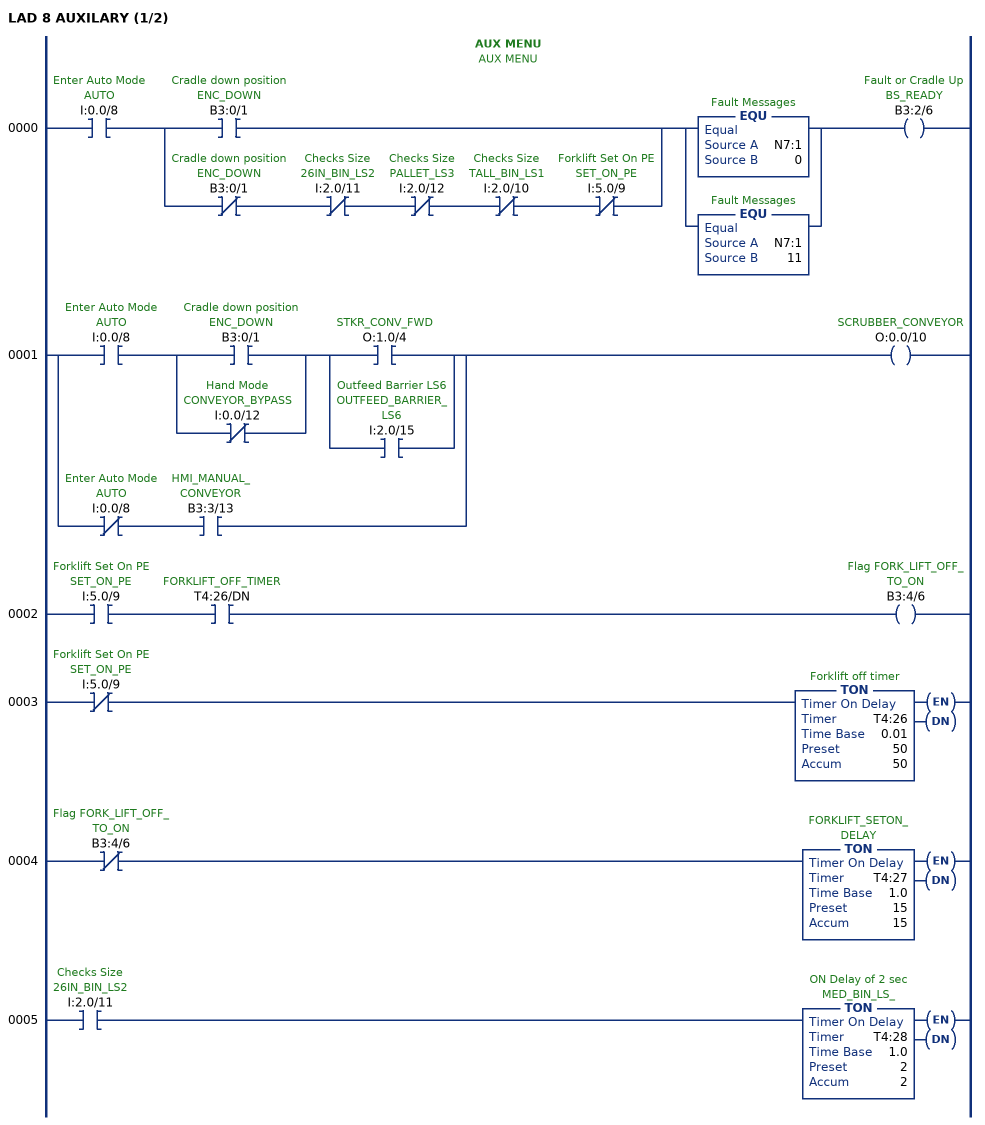
% Rung: 0 %
% TITLE: AUX MENU %
% AUX MENU %
SOR XIC I:0.0/8 BST XIC B3:0/1 NXB XIO B3:0/1 XIO I:2.0/11 XIO I:2.0/12 XIO I:2.0/10 XIO I:5.0/9 BND BST EQU N7:1 0 NXB EQU N7:1 11 BND OTE B3:2/6 EOR
%   I:0.0/8  AUTO  "Enter Auto Mode" %
%   B3:0/1  ENC_DOWN  "Cradle down position" %
%   I:2.0/11  26IN_BIN_LS2  "Checks Size" %
%   I:2.0/12  PALLET_LS3  "Checks Size" %
%   I:2.0/10  TALL_BIN_LS1  "Checks Size" %
%   I:5.0/9  SET_ON_PE  "Forklift Set On PE" %
%   N7:1  "Fault Messages" %
%   B3:2/6  BS_READY  "Fault or Cradle Up" %
% Rung: 1 %
SOR BST XIC I:0.0/8 BST XIC B3:0/1 NXB XIO I:0.0/12 BND BST XIC O:1.0/4 NXB XIC I:2.0/15 BND NXB XIO I:0.0/8 XIC B3:3/13 BND OTE O:0.0/10 EOR
%   I:0.0/8  AUTO  "Enter Auto Mode" %
%   B3:0/1  ENC_DOWN  "Cradle down position" %
%   I:0.0/12  CONVEYOR_BYPASS  "Hand Mode" %
%   O:1.0/4  STKR_CONV_FWD %
%   I:2.0/15  OUTFEED_BARRIER_LS6  "Outfeed Barrier LS6" %
%   B3:3/13  HMI_MANUAL_CONVEYOR %
%   O:0.0/10  SCRUBBER_CONVEYOR %
% Rung: 2 %
SOR XIC I:5.0/9 XIC T4:26/DN OTE B3:4/6 EOR
%   I:5.0/9  SET_ON_PE  "Forklift Set On PE" %
%   T4:26/DN  FORKLIFT_OFF_TIMER %
%   B3:4/6  FORK_LIFT_OFF_TO_ON  "Flag" %
% Rung: 3 %
SOR XIO I:5.0/9 TON T4:26 0.01 50 50 EOR
%   I:5.0/9  SET_ON_PE  "Forklift Set On PE" %
%   T4:26  "Forklift off timer" %
% Rung: 4 %
SOR XIO B3:4/6 TON T4:27 1.0 15 15 EOR
%   B3:4/6  FORK_LIFT_OFF_TO_ON  "Flag" %
%   T4:27  FORKLIFT_SETON_DELAY %
% Rung: 5 %
SOR XIC I:2.0/11 TON T4:28 1.0 2 2 EOR
%   I:2.0/11  26IN_BIN_LS2  "Checks Size" %
%   T4:28  MED_BIN_LS_  "ON Delay of 2 sec" %

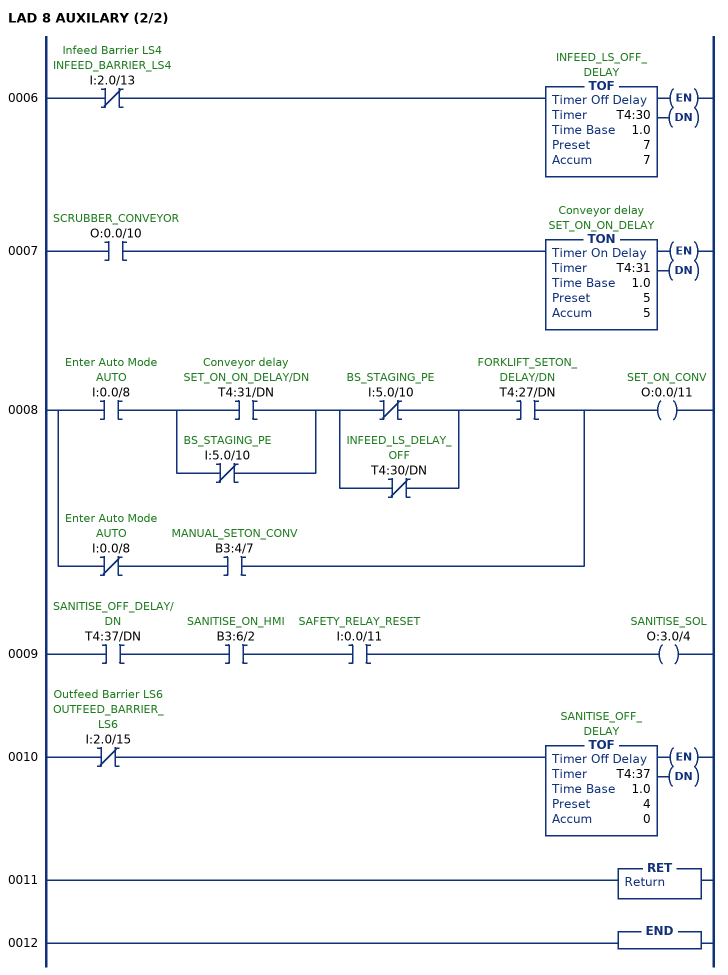
% Rung: 6 %
SOR XIO I:2.0/13 TOF T4:30 1.0 7 7 EOR
%   I:2.0/13  INFEED_BARRIER_LS4  "Infeed Barrier LS4" %
%   T4:30  INFEED_LS_OFF_DELAY %
% Rung: 7 %
SOR XIC O:0.0/10 TON T4:31 1.0 5 5 EOR
%   O:0.0/10  SCRUBBER_CONVEYOR %
%   T4:31  SET_ON_ON_DELAY  "Conveyor delay" %
% Rung: 8 %
SOR BST XIC I:0.0/8 BST XIC T4:31/DN NXB XIO I:5.0/10 BND BST XIO I:5.0/10 NXB XIO T4:30/DN BND XIC T4:27/DN NXB XIO I:0.0/8 XIC B3:4/7 BND OTE O:0.0/11 EOR
%   I:0.0/8  AUTO  "Enter Auto Mode" %
%   T4:31  SET_ON_ON_DELAY  "Conveyor delay" %
%   I:5.0/10  BS_STAGING_PE %
%   T4:30/DN  INFEED_LS_DELAY_OFF %
%   T4:27  FORKLIFT_SETON_DELAY %
%   B3:4/7  MANUAL_SETON_CONV %
%   O:0.0/11  SET_ON_CONV %
% Rung: 9 %
SOR XIC T4:37/DN XIC B3:6/2 XIC I:0.0/11 OTE O:3.0/4 EOR
%   T4:37  SANITISE_OFF_DELAY %
%   B3:6/2  SANITISE_ON_HMI %
%   I:0.0/11  SAFETY_RELAY_RESET %
%   O:3.0/4  SANITISE_SOL %
% Rung: 10 %
SOR XIO I:2.0/15 TOF T4:37 1.0 4 0 EOR
%   I:2.0/15  OUTFEED_BARRIER_LS6  "Outfeed Barrier LS6" %
%   T4:37  SANITISE_OFF_DELAY %
% Rung: 11 %
SOR RET EOR
% Rung: 12 %
SOR END EOR

LADDER 9 "FAULTS"
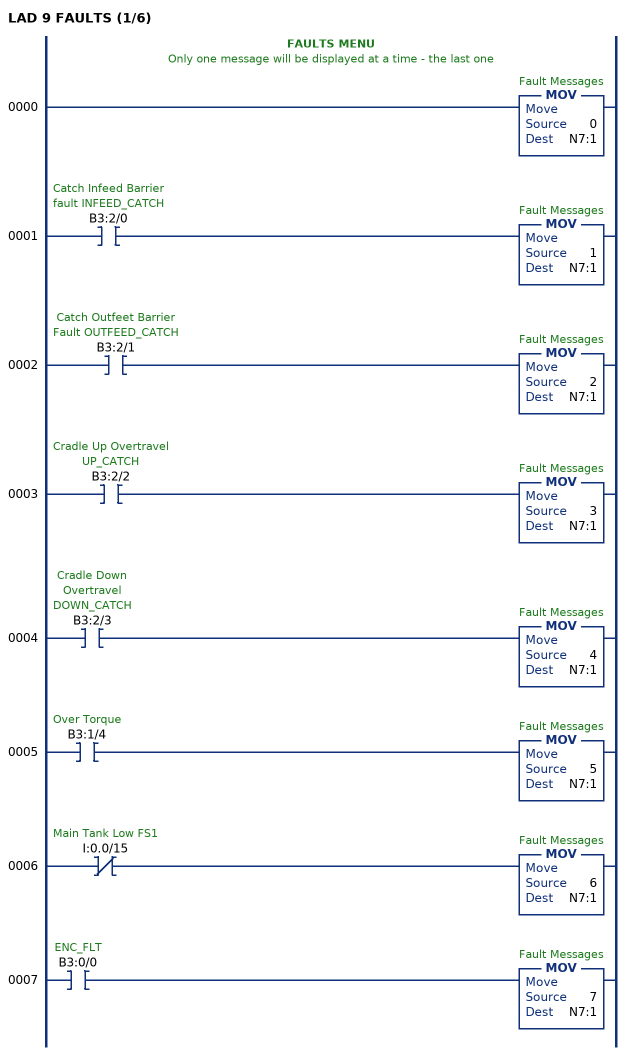
% Rung: 0 %
% TITLE: FAULTS MENU %
% Only one message will be displayed at a time - the last one %
SOR MOV 0 N7:1 EOR
%   N7:1  "Fault Messages" %
% Rung: 1 %
SOR XIC B3:2/0 MOV 1 N7:1 EOR
%   B3:2/0  INFEED_CATCH  "Catch Infeed Barrier fault" %
%   N7:1  "Fault Messages" %
% Rung: 2 %
SOR XIC B3:2/1 MOV 2 N7:1 EOR
%   B3:2/1  OUTFEED_CATCH  "Catch Outfeet Barrier Fault" %
%   N7:1  "Fault Messages" %
% Rung: 3 %
SOR XIC B3:2/2 MOV 3 N7:1 EOR
%   B3:2/2  UP_CATCH  "Cradle Up Overtravel" %
%   N7:1  "Fault Messages" %
% Rung: 4 %
SOR XIC B3:2/3 MOV 4 N7:1 EOR
%   B3:2/3  DOWN_CATCH  "Cradle Down Overtravel" %
%   N7:1  "Fault Messages" %
% Rung: 5 %
SOR XIC B3:1/4 MOV 5 N7:1 EOR
%   B3:1/4  "Over Torque" %
%   N7:1  "Fault Messages" %
% Rung: 6 %
SOR XIO I:0.0/15 MOV 6 N7:1 EOR
%   I:0.0/15  FS1  "Main Tank Low" %
%   N7:1  "Fault Messages" %
% Rung: 7 %
SOR XIC B3:0/0 MOV 7 N7:1 EOR
%   B3:0/0  ENC_FLT %
%   N7:1  "Fault Messages" %

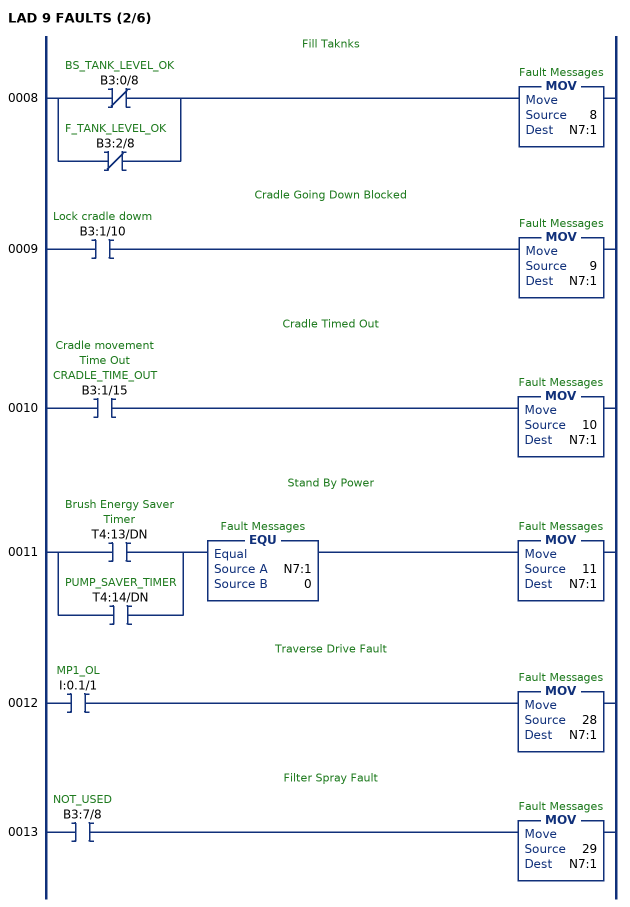
% Rung: 8 %
% Fill Taknks %
SOR BST XIO B3:0/8 NXB XIO B3:2/8 BND MOV 8 N7:1 EOR
%   B3:0/8  BS_TANK_LEVEL_OK %
%   B3:2/8  F_TANK_LEVEL_OK %
%   N7:1  "Fault Messages" %
% Rung: 9 %
% Cradle Going Down Blocked %
SOR XIC B3:1/10 MOV 9 N7:1 EOR
%   B3:1/10  "Lock cradle dowm" %
%   N7:1  "Fault Messages" %
% Rung: 10 %
% Cradle Timed Out %
SOR XIC B3:1/15 MOV 10 N7:1 EOR
%   B3:1/15  CRADLE_TIME_OUT  "Cradle movement Time Out" %
%   N7:1  "Fault Messages" %
% Rung: 11 %
% Stand By Power %
SOR BST XIC T4:13/DN NXB XIC T4:14/DN BND EQU N7:1 0 MOV 11 N7:1 EOR
%   T4:13  "Brush Energy Saver Timer" %
%   T4:14/DN  PUMP_SAVER_TIMER %
%   N7:1  "Fault Messages" %
% Rung: 12 %
% Traverse Drive Fault %
SOR XIC I:0.1/1 MOV 28 N7:1 EOR
%   I:0.1/1  MP1_OL %
%   N7:1  "Fault Messages" %
% Rung: 13 %
% Filter Spray Fault %
SOR XIC B3:7/8 MOV 29 N7:1 EOR
%   B3:7/8  NOT_USED %
%   N7:1  "Fault Messages" %

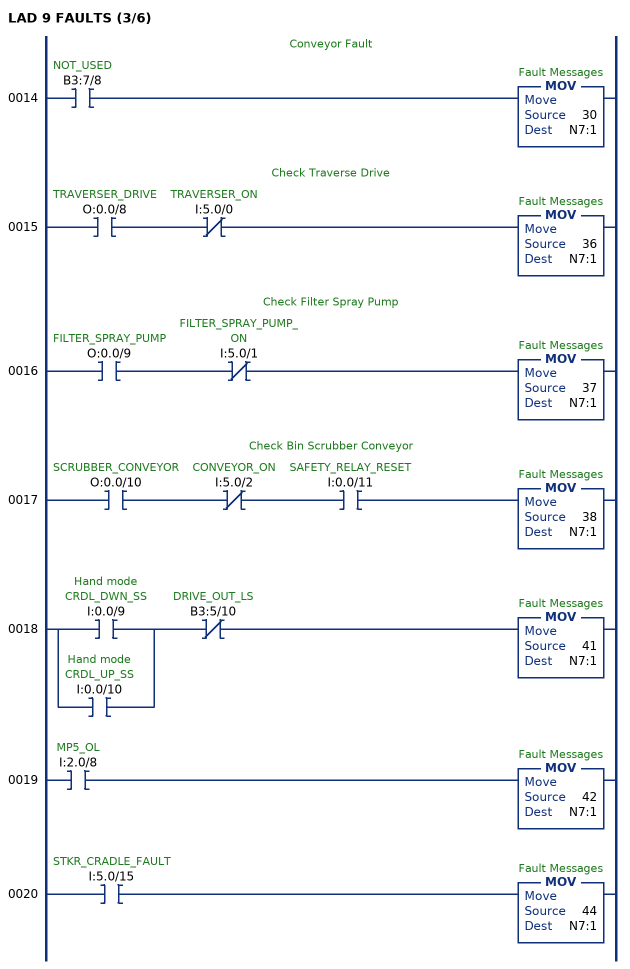
% Rung: 14 %
% Conveyor Fault %
SOR XIC B3:7/8 MOV 30 N7:1 EOR
%   B3:7/8  NOT_USED %
%   N7:1  "Fault Messages" %
% Rung: 15 %
% Check Traverse Drive %
SOR XIC O:0.0/8 XIO I:5.0/0 MOV 36 N7:1 EOR
%   O:0.0/8  TRAVERSER_DRIVE %
%   I:5.0/0  TRAVERSER_ON %
%   N7:1  "Fault Messages" %
% Rung: 16 %
% Check Filter Spray Pump %
SOR XIC O:0.0/9 XIO I:5.0/1 MOV 37 N7:1 EOR
%   O:0.0/9  FILTER_SPRAY_PUMP %
%   I:5.0/1  FILTER_SPRAY_PUMP_ON %
%   N7:1  "Fault Messages" %
% Rung: 17 %
% Check Bin Scrubber Conveyor %
SOR XIC O:0.0/10 XIO I:5.0/2 XIC I:0.0/11 MOV 38 N7:1 EOR
%   O:0.0/10  SCRUBBER_CONVEYOR %
%   I:5.0/2  CONVEYOR_ON %
%   I:0.0/11  SAFETY_RELAY_RESET %
%   N7:1  "Fault Messages" %
% Rung: 18 %
SOR BST XIC I:0.0/9 NXB XIC I:0.0/10 BND XIO B3:5/10 MOV 41 N7:1 EOR
%   I:0.0/9  CRDL_DWN_SS  "Hand mode" %
%   I:0.0/10  CRDL_UP_SS  "Hand mode" %
%   B3:5/10  DRIVE_OUT_LS %
%   N7:1  "Fault Messages" %
% Rung: 19 %
SOR XIC I:2.0/8 MOV 42 N7:1 EOR
%   I:2.0/8  MP5_OL %
%   N7:1  "Fault Messages" %
% Rung: 20 %
SOR XIC I:5.0/15 MOV 44 N7:1 EOR
%   I:5.0/15  STKR_CRADLE_FAULT %
%   N7:1  "Fault Messages" %

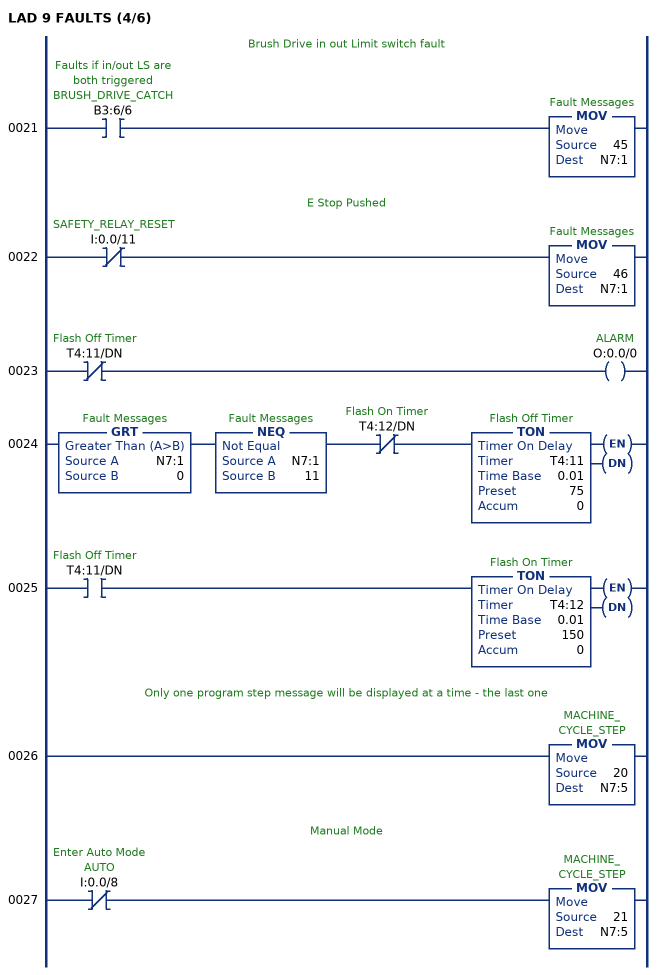
% Rung: 21 %
% Brush Drive in out Limit switch fault %
SOR XIC B3:6/6 MOV 45 N7:1 EOR
%   B3:6/6  BRUSH_DRIVE_CATCH  "Faults if in/out LS are both triggered" %
%   N7:1  "Fault Messages" %
% Rung: 22 %
% E Stop Pushed %
SOR XIO I:0.0/11 MOV 46 N7:1 EOR
%   I:0.0/11  SAFETY_RELAY_RESET %
%   N7:1  "Fault Messages" %
% Rung: 23 %
SOR XIO T4:11/DN OTE O:0.0/0 EOR
%   T4:11  "Flash Off Timer" %
%   O:0.0/0  ALARM %
% Rung: 24 %
SOR GRT N7:1 0 NEQ N7:1 11 XIO T4:12/DN TON T4:11 0.01 75 0 EOR
%   N7:1  "Fault Messages" %
%   T4:12  "Flash On Timer" %
%   T4:11  "Flash Off Timer" %
% Rung: 25 %
SOR XIC T4:11/DN TON T4:12 0.01 150 0 EOR
%   T4:11  "Flash Off Timer" %
%   T4:12  "Flash On Timer" %
% Rung: 26 %
% Only one program step message will be displayed at a time - the last one %
SOR MOV 20 N7:5 EOR
%   N7:5  MACHINE_CYCLE_STEP %
% Rung: 27 %
% Manual Mode %
SOR XIO I:0.0/8 MOV 21 N7:5 EOR
%   I:0.0/8  AUTO  "Enter Auto Mode" %
%   N7:5  MACHINE_CYCLE_STEP %

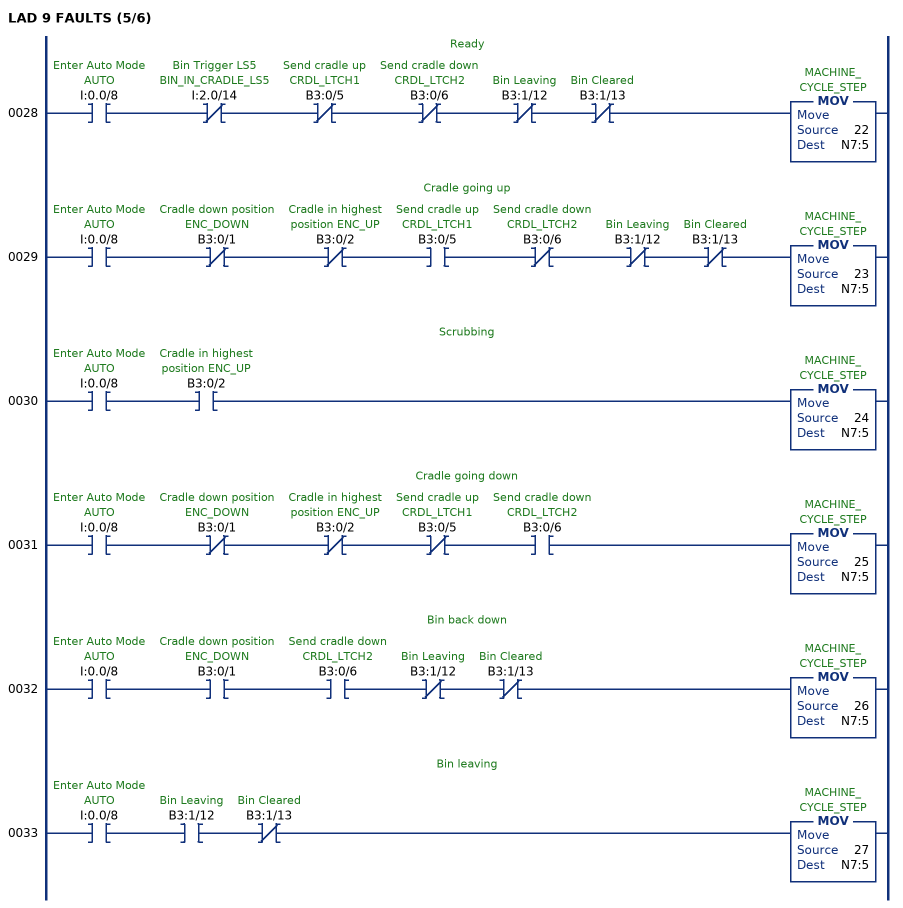
% Rung: 28 %
% Ready %
SOR XIC I:0.0/8 XIO I:2.0/14 XIO B3:0/5 XIO B3:0/6 XIO B3:1/12 XIO B3:1/13 MOV 22 N7:5 EOR
%   I:0.0/8  AUTO  "Enter Auto Mode" %
%   I:2.0/14  BIN_IN_CRADLE_LS5  "Bin Trigger LS5" %
%   B3:0/5  CRDL_LTCH1  "Send cradle up" %
%   B3:0/6  CRDL_LTCH2  "Send cradle down" %
%   B3:1/12  "Bin Leaving" %
%   B3:1/13  "Bin Cleared" %
%   N7:5  MACHINE_CYCLE_STEP %
% Rung: 29 %
% Cradle going up %
SOR XIC I:0.0/8 XIO B3:0/1 XIO B3:0/2 XIC B3:0/5 XIO B3:0/6 XIO B3:1/12 XIO B3:1/13 MOV 23 N7:5 EOR
%   I:0.0/8  AUTO  "Enter Auto Mode" %
%   B3:0/1  ENC_DOWN  "Cradle down position" %
%   B3:0/2  ENC_UP  "Cradle in highest position" %
%   B3:0/5  CRDL_LTCH1  "Send cradle up" %
%   B3:0/6  CRDL_LTCH2  "Send cradle down" %
%   B3:1/12  "Bin Leaving" %
%   B3:1/13  "Bin Cleared" %
%   N7:5  MACHINE_CYCLE_STEP %
% Rung: 30 %
% Scrubbing %
SOR XIC I:0.0/8 XIC B3:0/2 MOV 24 N7:5 EOR
%   I:0.0/8  AUTO  "Enter Auto Mode" %
%   B3:0/2  ENC_UP  "Cradle in highest position" %
%   N7:5  MACHINE_CYCLE_STEP %
% Rung: 31 %
% Cradle going down %
SOR XIC I:0.0/8 XIO B3:0/1 XIO B3:0/2 XIO B3:0/5 XIC B3:0/6 MOV 25 N7:5 EOR
%   I:0.0/8  AUTO  "Enter Auto Mode" %
%   B3:0/1  ENC_DOWN  "Cradle down position" %
%   B3:0/2  ENC_UP  "Cradle in highest position" %
%   B3:0/5  CRDL_LTCH1  "Send cradle up" %
%   B3:0/6  CRDL_LTCH2  "Send cradle down" %
%   N7:5  MACHINE_CYCLE_STEP %
% Rung: 32 %
% Bin back down %
SOR XIC I:0.0/8 XIC B3:0/1 XIC B3:0/6 XIO B3:1/12 XIO B3:1/13 MOV 26 N7:5 EOR
%   I:0.0/8  AUTO  "Enter Auto Mode" %
%   B3:0/1  ENC_DOWN  "Cradle down position" %
%   B3:0/6  CRDL_LTCH2  "Send cradle down" %
%   B3:1/12  "Bin Leaving" %
%   B3:1/13  "Bin Cleared" %
%   N7:5  MACHINE_CYCLE_STEP %
% Rung: 33 %
% Bin leaving %
SOR XIC I:0.0/8 XIC B3:1/12 XIO B3:1/13 MOV 27 N7:5 EOR
%   I:0.0/8  AUTO  "Enter Auto Mode" %
%   B3:1/12  "Bin Leaving" %
%   B3:1/13  "Bin Cleared" %
%   N7:5  MACHINE_CYCLE_STEP %

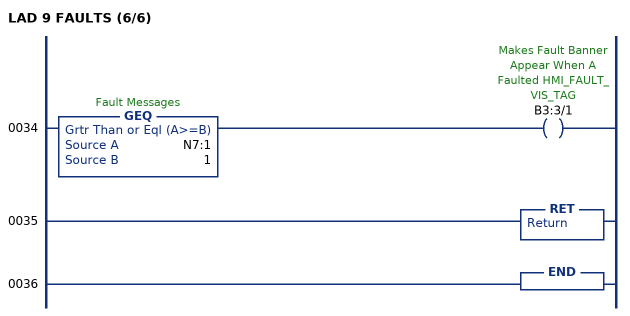
% Rung: 34 %
SOR GEQ N7:1 1 OTE B3:3/1 EOR
%   N7:1  "Fault Messages" %
%   B3:3/1  HMI_FAULT_VIS_TAG  "Makes Fault Banner Appear When A Faulted" %
% Rung: 35 %
SOR RET EOR
% Rung: 36 %
SOR END EOR

LADDER 10 "PID ANALOG"    % Scaling %
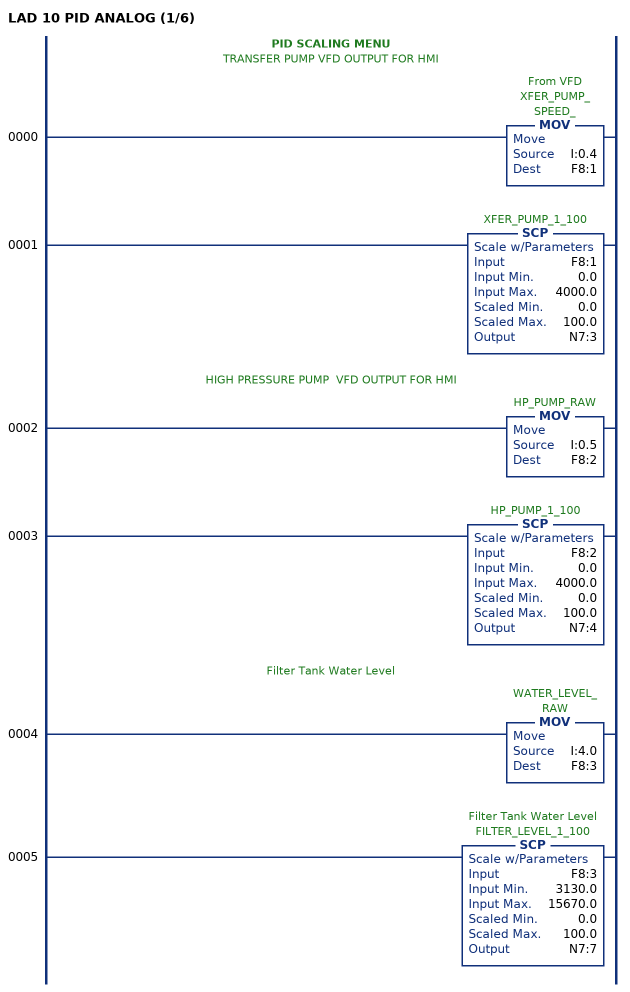
% Rung: 0 %
% TITLE: PID SCALING MENU %
% TRANSFER PUMP VFD OUTPUT FOR HMI %
SOR MOV I:0.4 F8:1 EOR
%   I:0.4  TRANSFER_PUMP_SPEED  "0/10v" %
%   F8:1  XFER_PUMP_SPEED_  "From VFD" %
% Rung: 1 %
SOR SCP F8:1 0.0 4000.0 0.0 100.0 N7:3 EOR
%   F8:1  XFER_PUMP_SPEED_  "From VFD" %
%   N7:3  XFER_PUMP_1_100 %
% Rung: 2 %
% HIGH PRESSURE PUMP  VFD OUTPUT FOR HMI %
SOR MOV I:0.5 F8:2 EOR
%   I:0.5  HP_PUMP_SPEED  "0/10v" %
%   F8:2  HP_PUMP_RAW %
% Rung: 3 %
SOR SCP F8:2 0.0 4000.0 0.0 100.0 N7:4 EOR
%   F8:2  HP_PUMP_RAW %
%   N7:4  HP_PUMP_1_100 %
% Rung: 4 %
% Filter Tank Water Level %
SOR MOV I:4.0 F8:3 EOR
%   I:4.0  XFER_TANK_LEVEL  "Raw Value" %
%   F8:3  WATER_LEVEL_RAW %
% Rung: 5 %
SOR SCP F8:3 3130.0 15670.0 0.0 100.0 N7:7 EOR
%   F8:3  WATER_LEVEL_RAW %
%   N7:7  FILTER_LEVEL_1_100  "Filter Tank Water Level" %

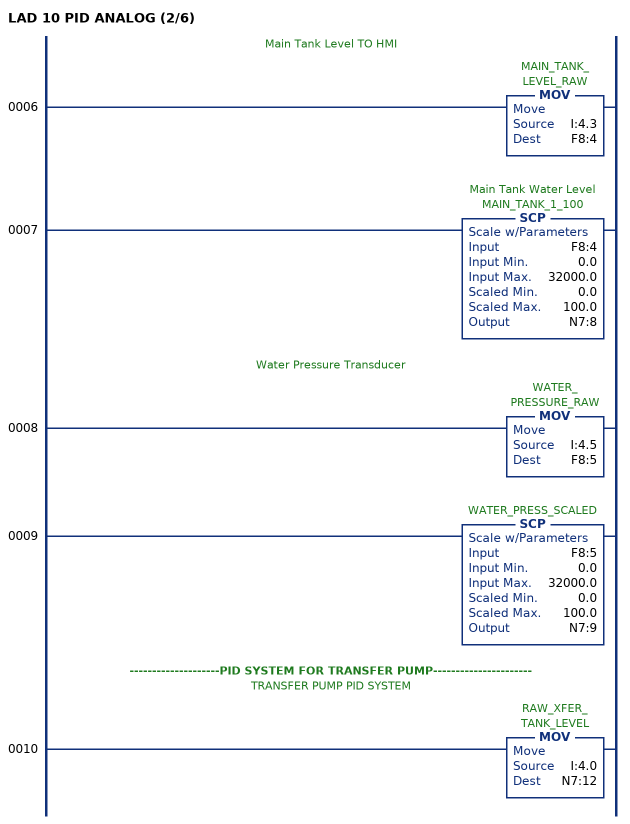
% Rung: 6 %
% Main Tank Level TO HMI %
SOR MOV I:4.3 F8:4 EOR
%   I:4.3  WATER_PRESSURE_SENS  "Pressure Sensor" %
%   F8:4  MAIN_TANK_LEVEL_RAW %
% Rung: 7 %
SOR SCP F8:4 0.0 32000.0 0.0 100.0 N7:8 EOR
%   F8:4  MAIN_TANK_LEVEL_RAW %
%   N7:8  MAIN_TANK_1_100  "Main Tank Water Level" %
% Rung: 8 %
% Water Pressure Transducer %
SOR MOV I:4.5 F8:5 EOR
%   F8:5  WATER_PRESSURE_RAW %
% Rung: 9 %
SOR SCP F8:5 0.0 32000.0 0.0 100.0 N7:9 EOR
%   F8:5  WATER_PRESSURE_RAW %
%   N7:9  WATER_PRESS_SCALED %
% Rung: 10 %
% TITLE: --------------------PID SYSTEM FOR TRANSFER PUMP---------------------- %
% TRANSFER PUMP PID SYSTEM %
SOR MOV I:4.0 N7:12 EOR
%   I:4.0  XFER_TANK_LEVEL  "Raw Value" %
%   N7:12  RAW_XFER_TANK_LEVEL %

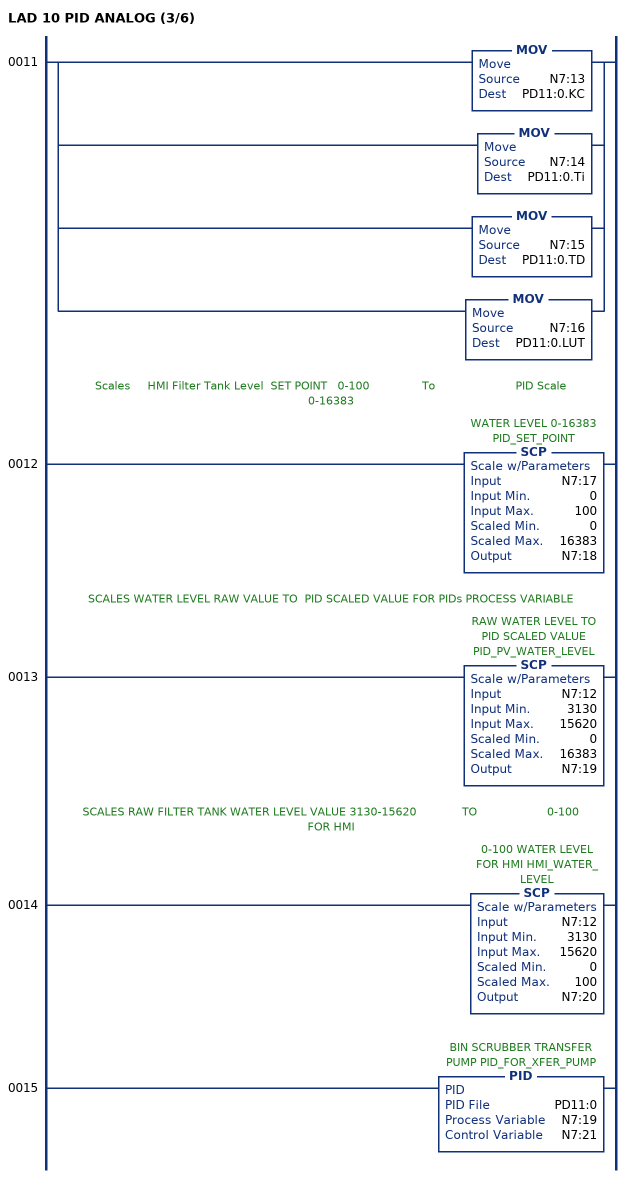
% Rung: 11 %
SOR BST MOV N7:13 PD11:0.KC NXB BST MOV N7:14 PD11:0.Ti NXB BST MOV N7:15 PD11:0.TD NXB MOV N7:16 PD11:0.LUT BND BND BND EOR
%   N7:13  KC_ %
%   N7:14  TI %
%   N7:15  TD %
%   N7:16  LUT %
% Rung: 12 %
% Scales     HMI Filter Tank Level  SET POINT   0-100               To                       PID Scale    0-16383 %
SOR SCP N7:17 0 100 0 16383 N7:18 EOR
%   N7:17  HMI_WATER_LEVEL_SP  "0-100" %
%   N7:18  PID_SET_POINT  "WATER LEVEL 0-16383" %
% Rung: 13 %
% SCALES WATER LEVEL RAW VALUE TO  PID SCALED VALUE FOR PIDs PROCESS VARIABLE %
SOR SCP N7:12 3130 15620 0 16383 N7:19 EOR
%   N7:12  RAW_XFER_TANK_LEVEL %
%   N7:19  PID_PV_WATER_LEVEL  "RAW WATER LEVEL TO PID SCALED VALUE" %
% Rung: 14 %
% SCALES RAW FILTER TANK WATER LEVEL VALUE 3130-15620             TO                    0-100  FOR HMI %
SOR SCP N7:12 3130 15620 0 100 N7:20 EOR
%   N7:12  RAW_XFER_TANK_LEVEL %
%   N7:20  HMI_WATER_LEVEL  "0-100 WATER LEVEL FOR HMI" %
% Rung: 15 %
SOR PID PD11:0 N7:19 N7:21 EOR
%   PD11:0  PID_FOR_XFER_PUMP  "BIN SCRUBBER TRANSFER PUMP" %
%   N7:19  PID_PV_WATER_LEVEL  "RAW WATER LEVEL TO PID SCALED VALUE" %
%   N7:21  PID_OUTPUT_RAW  "0-16383" %

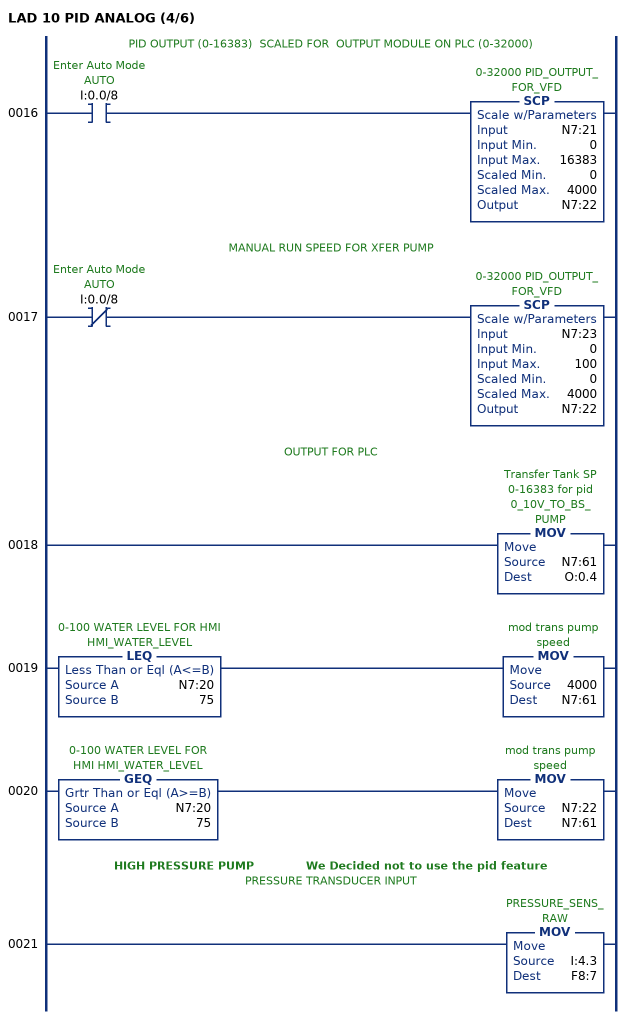
% Rung: 16 %
% PID OUTPUT (0-16383)  SCALED FOR  OUTPUT MODULE ON PLC (0-32000) %
SOR XIC I:0.0/8 SCP N7:21 0 16383 0 4000 N7:22 EOR
%   I:0.0/8  AUTO  "Enter Auto Mode" %
%   N7:21  PID_OUTPUT_RAW  "0-16383" %
%   N7:22  PID_OUTPUT_FOR_VFD  "0-32000" %
% Rung: 17 %
% MANUAL RUN SPEED FOR XFER PUMP %
SOR XIO I:0.0/8 SCP N7:23 0 100 0 4000 N7:22 EOR
%   I:0.0/8  AUTO  "Enter Auto Mode" %
%   N7:23  HMI_MANUAL_RUN %
%   N7:22  PID_OUTPUT_FOR_VFD  "0-32000" %
% Rung: 18 %
% OUTPUT FOR PLC %
SOR MOV N7:61 O:0.4 EOR
%   N7:61  "mod trans pump speed" %
%   O:0.4  0_10V_TO_BS_PUMP  "Transfer Tank SP 0-16383 for pid" %
% Rung: 19 %
SOR LEQ N7:20 75 MOV 4000 N7:61 EOR
%   N7:20  HMI_WATER_LEVEL  "0-100 WATER LEVEL FOR HMI" %
%   N7:61  "mod trans pump speed" %
% Rung: 20 %
SOR GEQ N7:20 75 MOV N7:22 N7:61 EOR
%   N7:20  HMI_WATER_LEVEL  "0-100 WATER LEVEL FOR HMI" %
%   N7:22  PID_OUTPUT_FOR_VFD  "0-32000" %
%   N7:61  "mod trans pump speed" %
% Rung: 21 %
% TITLE: HIGH PRESSURE PUMP             We Decided not to use the pid feature %
% PRESSURE TRANSDUCER INPUT %
SOR MOV I:4.3 F8:7 EOR
%   I:4.3  WATER_PRESSURE_SENS  "Pressure Sensor" %
%   F8:7  PRESSURE_SENS_RAW %

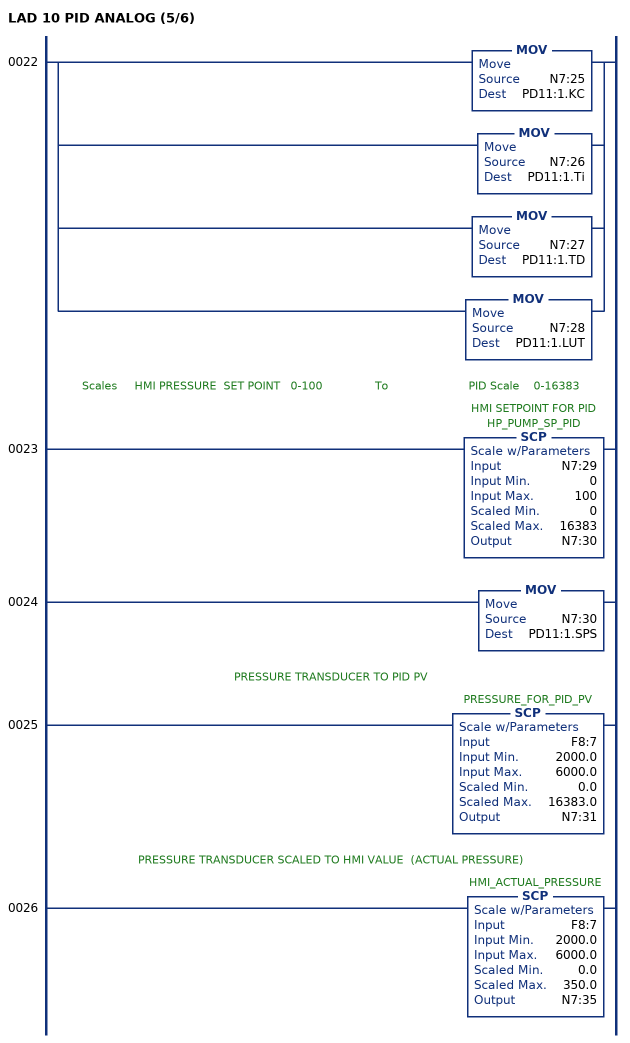
% Rung: 22 %
SOR BST MOV N7:25 PD11:1.KC NXB BST MOV N7:26 PD11:1.Ti NXB BST MOV N7:27 PD11:1.TD NXB MOV N7:28 PD11:1.LUT BND BND BND EOR
%   N7:25  HP_KC_SP %
%   N7:26  HP_TI_SP %
%   N7:27  HP_TD_SP %
%   N7:28  HP_LUT_SP %
% Rung: 23 %
% Scales     HMI PRESSURE  SET POINT   0-100               To                       PID Scale    0-16383 %
SOR SCP N7:29 0 100 0 16383 N7:30 EOR
%   N7:29  HMI_PRESSURE_SP  "HP PUMP PRESSURE SP" %
%   N7:30  HP_PUMP_SP_PID  "HMI SETPOINT FOR PID" %
% Rung: 24 %
SOR MOV N7:30 PD11:1.SPS EOR
%   N7:30  HP_PUMP_SP_PID  "HMI SETPOINT FOR PID" %
% Rung: 25 %
% PRESSURE TRANSDUCER TO PID PV %
SOR SCP F8:7 2000.0 6000.0 0.0 16383.0 N7:31 EOR
%   F8:7  PRESSURE_SENS_RAW %
%   N7:31  PRESSURE_FOR_PID_PV %
% Rung: 26 %
% PRESSURE TRANSDUCER SCALED TO HMI VALUE  (ACTUAL PRESSURE) %
SOR SCP F8:7 2000.0 6000.0 0.0 350.0 N7:35 EOR
%   F8:7  PRESSURE_SENS_RAW %
%   N7:35  HMI_ACTUAL_PRESSURE %

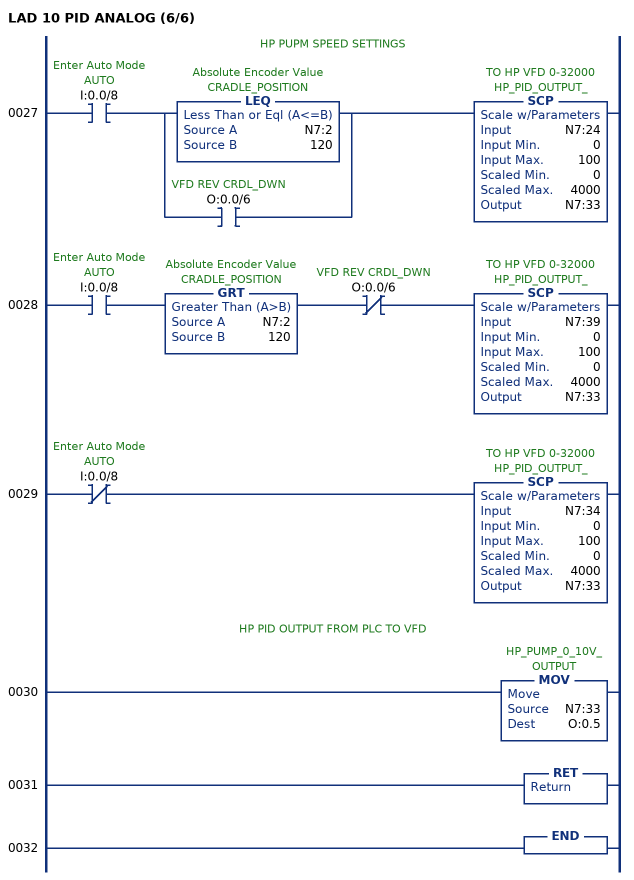
% Rung: 27 %
% HP PUPM SPEED SETTINGS %
SOR XIC I:0.0/8 BST LEQ N7:2 120 NXB XIC O:0.0/6 BND SCP N7:24 0 100 0 4000 N7:33 EOR
%   I:0.0/8  AUTO  "Enter Auto Mode" %
%   N7:2  CRADLE_POSITION  "Absolute Encoder Value" %
%   O:0.0/6  CRDL_DWN  "VFD REV" %
%   N7:24  HP_PUMP_SP  "HMI SP" %
%   N7:33  HP_PID_OUTPUT_  "TO HP VFD 0-32000" %
% Rung: 28 %
SOR XIC I:0.0/8 GRT N7:2 120 XIO O:0.0/6 SCP N7:39 0 100 0 4000 N7:33 EOR
%   I:0.0/8  AUTO  "Enter Auto Mode" %
%   N7:2  CRADLE_POSITION  "Absolute Encoder Value" %
%   O:0.0/6  CRDL_DWN  "VFD REV" %
%   N7:39  HP_SPEED_CRADLE_UP %
%   N7:33  HP_PID_OUTPUT_  "TO HP VFD 0-32000" %
% Rung: 29 %
SOR XIO I:0.0/8 SCP N7:34 0 100 0 4000 N7:33 EOR
%   I:0.0/8  AUTO  "Enter Auto Mode" %
%   N7:34  HMI_MANUAL_HP_SPEED  "HMI MANUAL RUN SPEED FOR HP PUMP" %
%   N7:33  HP_PID_OUTPUT_  "TO HP VFD 0-32000" %
% Rung: 30 %
% HP PID OUTPUT FROM PLC TO VFD %
SOR MOV N7:33 O:0.5 EOR
%   N7:33  HP_PID_OUTPUT_  "TO HP VFD 0-32000" %
%   O:0.5  HP_PUMP_0_10V_OUTPUT %
% Rung: 31 %
SOR RET EOR
% Rung: 32 %
SOR END EOR

LADDER 11 "BIN SIZING"    % Bin sizing Pallet, 26", Tall %
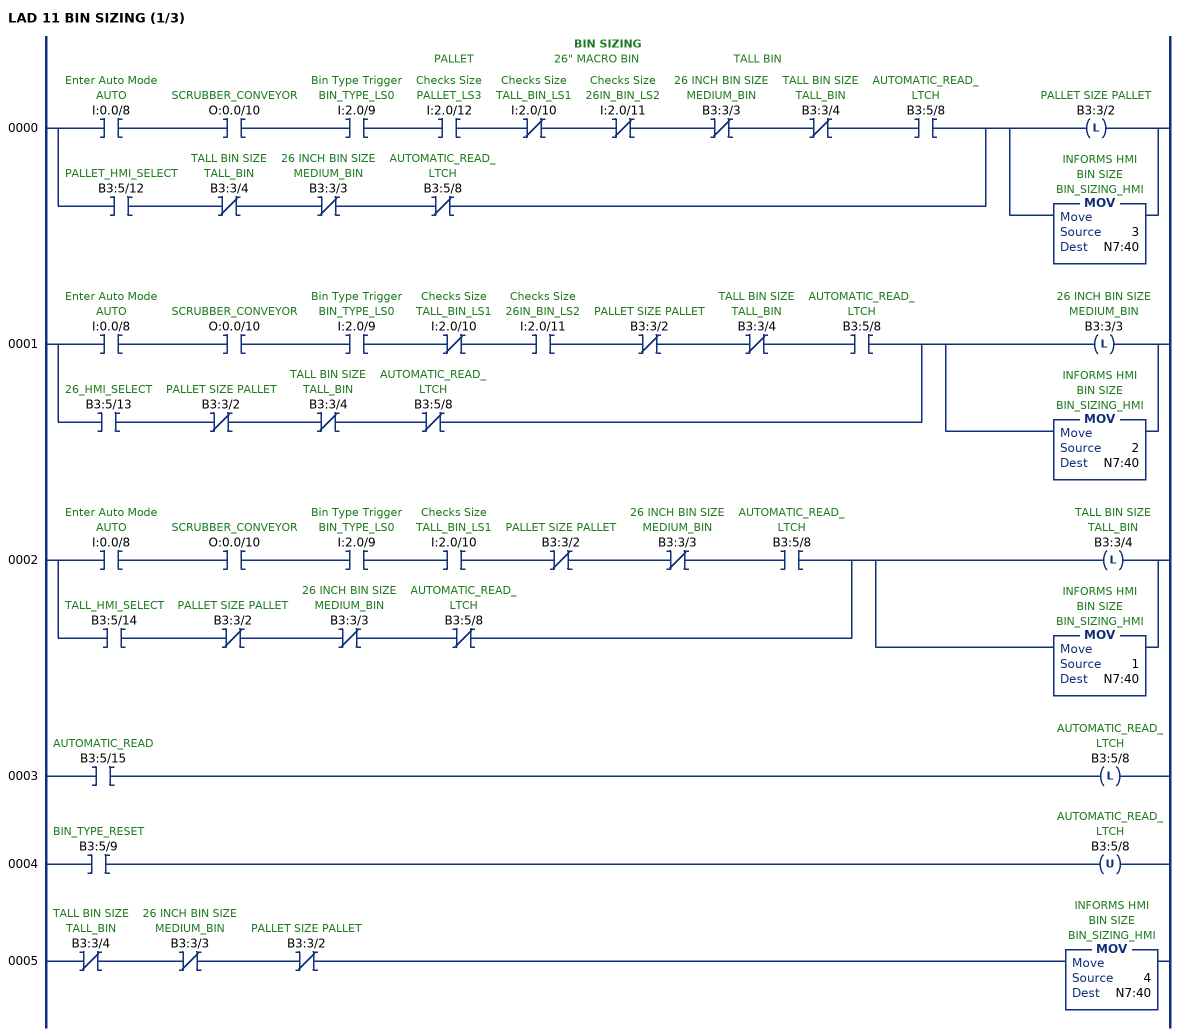
% Rung: 0 %
% TITLE: BIN SIZING %
% PALLET                       26" MACRO BIN                           TALL BIN %
SOR BST XIC I:0.0/8 XIC O:0.0/10 XIC I:2.0/9 XIC I:2.0/12 XIO I:2.0/10 XIO I:2.0/11 XIO B3:3/3 XIO B3:3/4 XIC B3:5/8 NXB XIC B3:5/12 XIO B3:3/4 XIO B3:3/3 XIO B3:5/8 BND BST OTL B3:3/2 NXB MOV 3 N7:40 BND EOR
%   I:0.0/8  AUTO  "Enter Auto Mode" %
%   O:0.0/10  SCRUBBER_CONVEYOR %
%   I:2.0/9  BIN_TYPE_LS0  "Bin Type Trigger" %
%   I:2.0/12  PALLET_LS3  "Checks Size" %
%   I:2.0/10  TALL_BIN_LS1  "Checks Size" %
%   I:2.0/11  26IN_BIN_LS2  "Checks Size" %
%   B3:3/3  MEDIUM_BIN  "26 INCH BIN SIZE" %
%   B3:3/4  TALL_BIN  "TALL BIN SIZE" %
%   B3:5/8  AUTOMATIC_READ_LTCH %
%   B3:5/12  PALLET_HMI_SELECT %
%   B3:3/2  PALLET  "PALLET SIZE" %
%   N7:40  BIN_SIZING_HMI  "INFORMS HMI BIN SIZE" %
% Rung: 1 %
SOR BST XIC I:0.0/8 XIC O:0.0/10 XIC I:2.0/9 XIO I:2.0/10 XIC I:2.0/11 XIO B3:3/2 XIO B3:3/4 XIC B3:5/8 NXB XIC B3:5/13 XIO B3:3/2 XIO B3:3/4 XIO B3:5/8 BND BST OTL B3:3/3 NXB MOV 2 N7:40 BND EOR
%   I:0.0/8  AUTO  "Enter Auto Mode" %
%   O:0.0/10  SCRUBBER_CONVEYOR %
%   I:2.0/9  BIN_TYPE_LS0  "Bin Type Trigger" %
%   I:2.0/10  TALL_BIN_LS1  "Checks Size" %
%   I:2.0/11  26IN_BIN_LS2  "Checks Size" %
%   B3:3/2  PALLET  "PALLET SIZE" %
%   B3:3/4  TALL_BIN  "TALL BIN SIZE" %
%   B3:5/8  AUTOMATIC_READ_LTCH %
%   B3:5/13  26_HMI_SELECT %
%   B3:3/3  MEDIUM_BIN  "26 INCH BIN SIZE" %
%   N7:40  BIN_SIZING_HMI  "INFORMS HMI BIN SIZE" %
% Rung: 2 %
SOR BST XIC I:0.0/8 XIC O:0.0/10 XIC I:2.0/9 XIC I:2.0/10 XIO B3:3/2 XIO B3:3/3 XIC B3:5/8 NXB XIC B3:5/14 XIO B3:3/2 XIO B3:3/3 XIO B3:5/8 BND BST OTL B3:3/4 NXB MOV 1 N7:40 BND EOR
%   I:0.0/8  AUTO  "Enter Auto Mode" %
%   O:0.0/10  SCRUBBER_CONVEYOR %
%   I:2.0/9  BIN_TYPE_LS0  "Bin Type Trigger" %
%   I:2.0/10  TALL_BIN_LS1  "Checks Size" %
%   B3:3/2  PALLET  "PALLET SIZE" %
%   B3:3/3  MEDIUM_BIN  "26 INCH BIN SIZE" %
%   B3:5/8  AUTOMATIC_READ_LTCH %
%   B3:5/14  TALL_HMI_SELECT %
%   B3:3/4  TALL_BIN  "TALL BIN SIZE" %
%   N7:40  BIN_SIZING_HMI  "INFORMS HMI BIN SIZE" %
% Rung: 3 %
SOR XIC B3:5/15 OTL B3:5/8 EOR
%   B3:5/15  AUTOMATIC_READ %
%   B3:5/8  AUTOMATIC_READ_LTCH %
% Rung: 4 %
SOR XIC B3:5/9 OTU B3:5/8 EOR
%   B3:5/9  BIN_TYPE_RESET %
%   B3:5/8  AUTOMATIC_READ_LTCH %
% Rung: 5 %
SOR XIO B3:3/4 XIO B3:3/3 XIO B3:3/2 MOV 4 N7:40 EOR
%   B3:3/4  TALL_BIN  "TALL BIN SIZE" %
%   B3:3/3  MEDIUM_BIN  "26 INCH BIN SIZE" %
%   B3:3/2  PALLET  "PALLET SIZE" %
%   N7:40  BIN_SIZING_HMI  "INFORMS HMI BIN SIZE" %

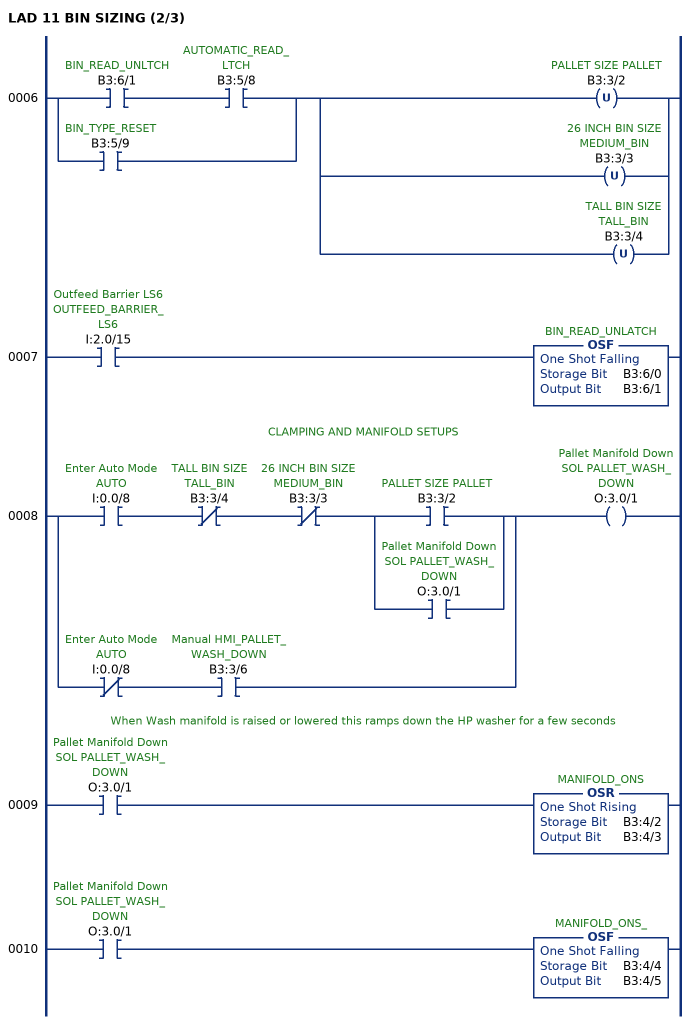
% Rung: 6 %
SOR BST XIC B3:6/1 XIC B3:5/8 NXB XIC B3:5/9 BND BST OTU B3:3/2 NXB BST OTU B3:3/3 NXB OTU B3:3/4 BND BND EOR
%   B3:6/1  BIN_READ_UNLTCH %
%   B3:5/8  AUTOMATIC_READ_LTCH %
%   B3:5/9  BIN_TYPE_RESET %
%   B3:3/2  PALLET  "PALLET SIZE" %
%   B3:3/3  MEDIUM_BIN  "26 INCH BIN SIZE" %
%   B3:3/4  TALL_BIN  "TALL BIN SIZE" %
% Rung: 7 %
SOR XIC I:2.0/15 OSF B3:6/0 B3:6/1 EOR
%   I:2.0/15  OUTFEED_BARRIER_LS6  "Outfeed Barrier LS6" %
%   B3:6/0  BIN_READ_UNLATCH %
%   B3:6/1  BIN_READ_UNLTCH %
% Rung: 8 %
% CLAMPING AND MANIFOLD SETUPS %
SOR BST XIC I:0.0/8 XIO B3:3/4 XIO B3:3/3 BST XIC B3:3/2 NXB XIC O:3.0/1 BND NXB XIO I:0.0/8 XIC B3:3/6 BND OTE O:3.0/1 EOR
%   I:0.0/8  AUTO  "Enter Auto Mode" %
%   B3:3/4  TALL_BIN  "TALL BIN SIZE" %
%   B3:3/3  MEDIUM_BIN  "26 INCH BIN SIZE" %
%   B3:3/2  PALLET  "PALLET SIZE" %
%   O:3.0/1  PALLET_WASH_DOWN  "Pallet Manifold Down SOL" %
%   B3:3/6  HMI_PALLET_WASH_DOWN  "Manual" %
% Rung: 9 %
% When Wash manifold is raised or lowered this ramps down the HP washer for a few seconds %
SOR XIC O:3.0/1 OSR B3:4/2 B3:4/3 EOR
%   O:3.0/1  PALLET_WASH_DOWN  "Pallet Manifold Down SOL" %
%   B3:4/2  MANIFOLD_ONS %
%   B3:4/3  MANIFOLD_DELAY_ONS %
% Rung: 10 %
SOR XIC O:3.0/1 OSF B3:4/4 B3:4/5 EOR
%   O:3.0/1  PALLET_WASH_DOWN  "Pallet Manifold Down SOL" %
%   B3:4/4  MANIFOLD_ONS_ %
%   B3:4/5  MANIFOLD_DELAY_ONS_ %

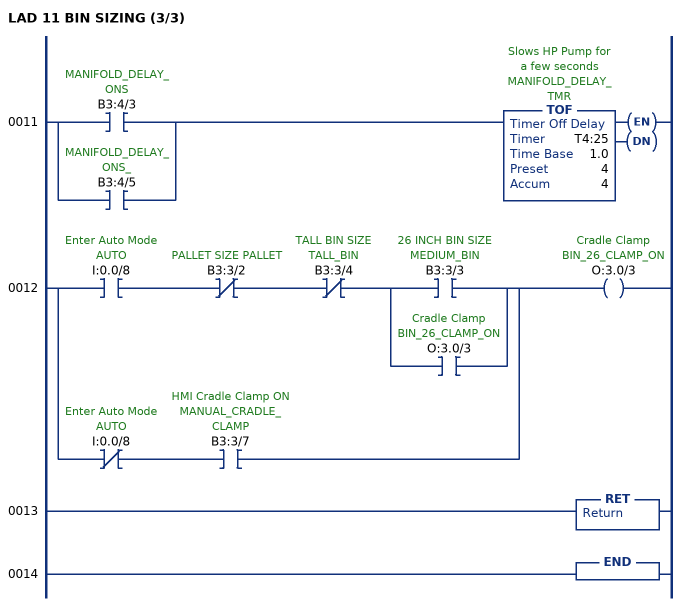
% Rung: 11 %
SOR BST XIC B3:4/3 NXB XIC B3:4/5 BND TOF T4:25 1.0 4 4 EOR
%   B3:4/3  MANIFOLD_DELAY_ONS %
%   B3:4/5  MANIFOLD_DELAY_ONS_ %
%   T4:25  MANIFOLD_DELAY_TMR  "Slows HP Pump for a few seconds" %
% Rung: 12 %
SOR BST XIC I:0.0/8 XIO B3:3/2 XIO B3:3/4 BST XIC B3:3/3 NXB XIC O:3.0/3 BND NXB XIO I:0.0/8 XIC B3:3/7 BND OTE O:3.0/3 EOR
%   I:0.0/8  AUTO  "Enter Auto Mode" %
%   B3:3/2  PALLET  "PALLET SIZE" %
%   B3:3/4  TALL_BIN  "TALL BIN SIZE" %
%   B3:3/3  MEDIUM_BIN  "26 INCH BIN SIZE" %
%   O:3.0/3  BIN_26_CLAMP_ON  "Cradle Clamp" %
%   B3:3/7  MANUAL_CRADLE_CLAMP  "HMI Cradle Clamp ON" %
% Rung: 13 %
SOR RET EOR
% Rung: 14 %
SOR END EOR

LADDER 12 "STACKER"
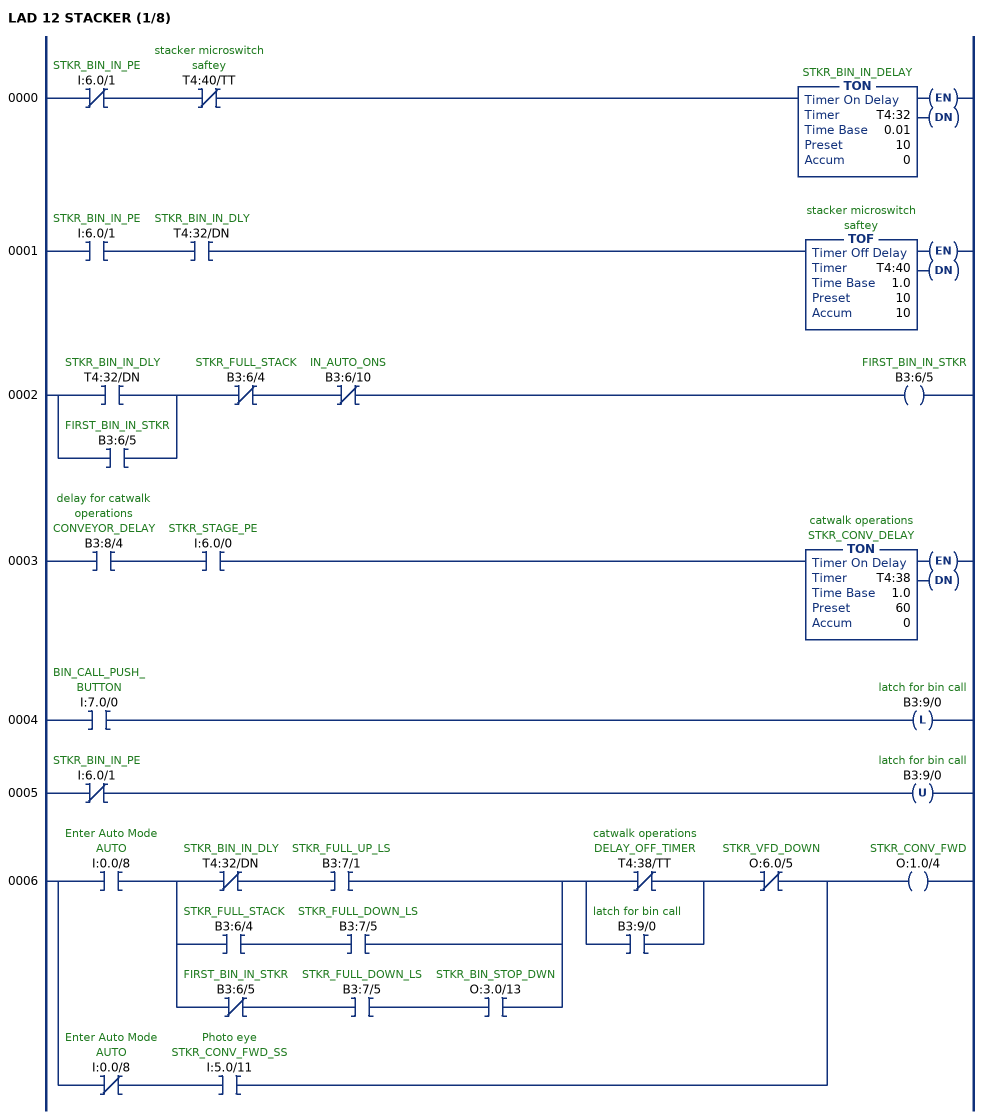
% Rung: 0 %
SOR XIO I:6.0/1 XIO T4:40/TT TON T4:32 0.01 10 0 EOR
%   I:6.0/1  STKR_BIN_IN_PE %
%   T4:40  "stacker microswitch saftey" %
%   T4:32  STKR_BIN_IN_DELAY %
% Rung: 1 %
SOR XIC I:6.0/1 XIC T4:32/DN TOF T4:40 1.0 10 10 EOR
%   I:6.0/1  STKR_BIN_IN_PE %
%   T4:32/DN  STKR_BIN_IN_DLY %
%   T4:40  "stacker microswitch saftey" %
% Rung: 2 %
SOR BST XIC T4:32/DN NXB XIC B3:6/5 BND XIO B3:6/4 XIO B3:6/10 OTE B3:6/5 EOR
%   T4:32/DN  STKR_BIN_IN_DLY %
%   B3:6/5  FIRST_BIN_IN_STKR %
%   B3:6/4  STKR_FULL_STACK %
%   B3:6/10  IN_AUTO_ONS %
% Rung: 3 %
SOR XIC B3:8/4 XIC I:6.0/0 TON T4:38 1.0 60 0 EOR
%   B3:8/4  CONVEYOR_DELAY  "delay for catwalk operations" %
%   I:6.0/0  STKR_STAGE_PE %
%   T4:38  STKR_CONV_DELAY  "catwalk operations" %
% Rung: 4 %
SOR XIC I:7.0/0 OTL B3:9/0 EOR
%   I:7.0/0  BIN_CALL_PUSH_BUTTON %
%   B3:9/0  "latch for bin call" %
% Rung: 5 %
SOR XIO I:6.0/1 OTU B3:9/0 EOR
%   I:6.0/1  STKR_BIN_IN_PE %
%   B3:9/0  "latch for bin call" %
% Rung: 6 %
SOR BST XIC I:0.0/8 BST XIO T4:32/DN XIC B3:7/1 NXB BST XIC B3:6/4 XIC B3:7/5 NXB XIO B3:6/5 XIC B3:7/5 XIC O:3.0/13 BND BND BST XIO T4:38/TT NXB XIC B3:9/0 BND XIO O:6.0/5 NXB XIO I:0.0/8 XIC I:5.0/11 BND OTE O:1.0/4 EOR
%   I:0.0/8  AUTO  "Enter Auto Mode" %
%   T4:32/DN  STKR_BIN_IN_DLY %
%   B3:7/1  STKR_FULL_UP_LS %
%   B3:6/4  STKR_FULL_STACK %
%   B3:7/5  STKR_FULL_DOWN_LS %
%   B3:6/5  FIRST_BIN_IN_STKR %
%   O:3.0/13  STKR_BIN_STOP_DWN %
%   T4:38/TT  DELAY_OFF_TIMER  "catwalk operations" %
%   B3:9/0  "latch for bin call" %
%   O:6.0/5  STKR_VFD_DOWN %
%   I:5.0/11  STKR_CONV_FWD_SS  "Photo eye" %
%   O:1.0/4  STKR_CONV_FWD %

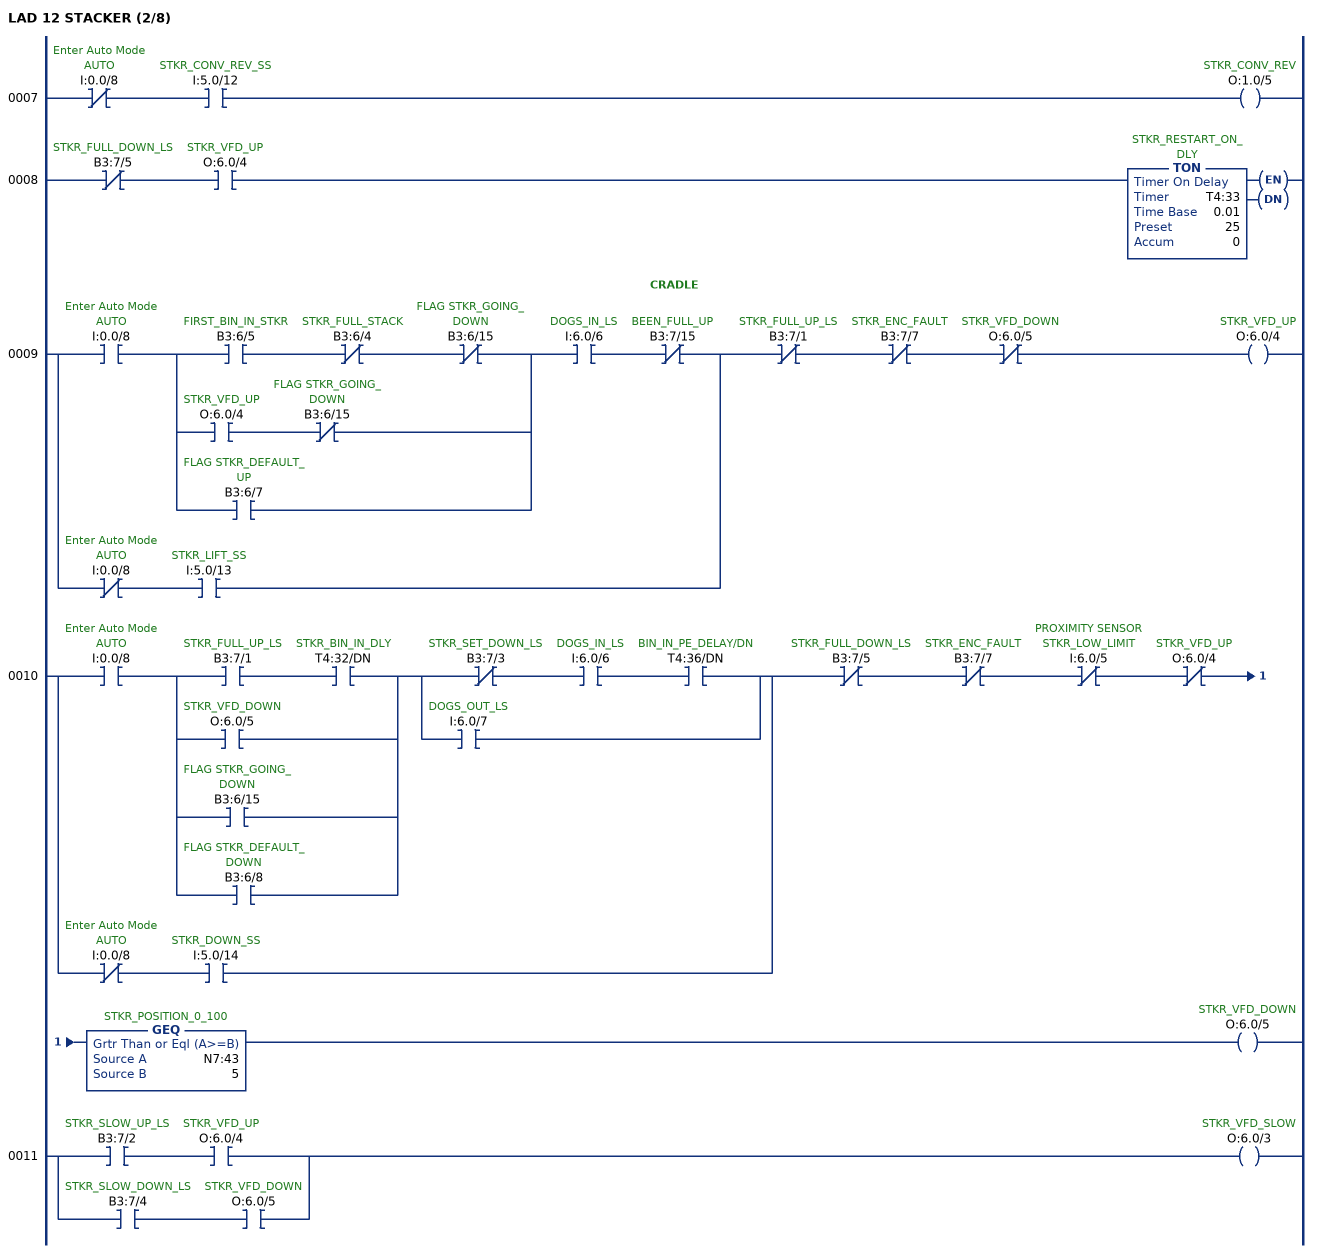
% Rung: 7 %
SOR XIO I:0.0/8 XIC I:5.0/12 OTE O:1.0/5 EOR
%   I:0.0/8  AUTO  "Enter Auto Mode" %
%   I:5.0/12  STKR_CONV_REV_SS %
%   O:1.0/5  STKR_CONV_REV %
% Rung: 8 %
SOR XIO B3:7/5 XIC O:6.0/4 TON T4:33 0.01 25 0 EOR
%   B3:7/5  STKR_FULL_DOWN_LS %
%   O:6.0/4  STKR_VFD_UP %
%   T4:33  STKR_RESTART_ON_DLY %
% Rung: 9 %
% TITLE: CRADLE %
SOR BST XIC I:0.0/8 BST XIC B3:6/5 XIO B3:6/4 XIO B3:6/15 NXB BST XIC O:6.0/4 XIO B3:6/15 NXB XIC B3:6/7 BND BND XIC I:6.0/6 XIO B3:7/15 NXB XIO I:0.0/8 XIC I:5.0/13 BND XIO B3:7/1 XIO B3:7/7 XIO O:6.0/5 OTE O:6.0/4 EOR
%   I:0.0/8  AUTO  "Enter Auto Mode" %
%   B3:6/5  FIRST_BIN_IN_STKR %
%   B3:6/4  STKR_FULL_STACK %
%   B3:6/15  STKR_GOING_DOWN  "FLAG" %
%   O:6.0/4  STKR_VFD_UP %
%   B3:6/7  STKR_DEFAULT_UP  "FLAG" %
%   I:6.0/6  DOGS_IN_LS %
%   B3:7/15  BEEN_FULL_UP %
%   I:5.0/13  STKR_LIFT_SS %
%   B3:7/1  STKR_FULL_UP_LS %
%   B3:7/7  STKR_ENC_FAULT %
%   O:6.0/5  STKR_VFD_DOWN %
% Rung: 10 %
SOR BST XIC I:0.0/8 BST XIC B3:7/1 XIC T4:32/DN NXB BST BST XIC O:6.0/5 NXB XIC B3:6/15 BND NXB XIC B3:6/8 BND BND BST XIO B3:7/3 XIC I:6.0/6 XIC T4:36/DN NXB XIC I:6.0/7 BND NXB XIO I:0.0/8 XIC I:5.0/14 BND XIO B3:7/5 XIO B3:7/7 XIO I:6.0/5 XIO O:6.0/4 GEQ N7:43 5 OTE O:6.0/5 EOR
%   I:0.0/8  AUTO  "Enter Auto Mode" %
%   B3:7/1  STKR_FULL_UP_LS %
%   T4:32/DN  STKR_BIN_IN_DLY %
%   O:6.0/5  STKR_VFD_DOWN %
%   B3:6/15  STKR_GOING_DOWN  "FLAG" %
%   B3:6/8  STKR_DEFAULT_DOWN  "FLAG" %
%   B3:7/3  STKR_SET_DOWN_LS %
%   I:6.0/6  DOGS_IN_LS %
%   T4:36  BIN_IN_PE_DELAY %
%   I:6.0/7  DOGS_OUT_LS %
%   I:5.0/14  STKR_DOWN_SS %
%   B3:7/5  STKR_FULL_DOWN_LS %
%   B3:7/7  STKR_ENC_FAULT %
%   I:6.0/5  STKR_LOW_LIMIT  "PROXIMITY SENSOR" %
%   O:6.0/4  STKR_VFD_UP %
%   N7:43  STKR_POSITION_0_100 %
% Rung: 11 %
SOR BST XIC B3:7/2 XIC O:6.0/4 NXB XIC B3:7/4 XIC O:6.0/5 BND OTE O:6.0/3 EOR
%   B3:7/2  STKR_SLOW_UP_LS %
%   O:6.0/4  STKR_VFD_UP %
%   B3:7/4  STKR_SLOW_DOWN_LS %
%   O:6.0/5  STKR_VFD_DOWN %
%   O:6.0/3  STKR_VFD_SLOW %

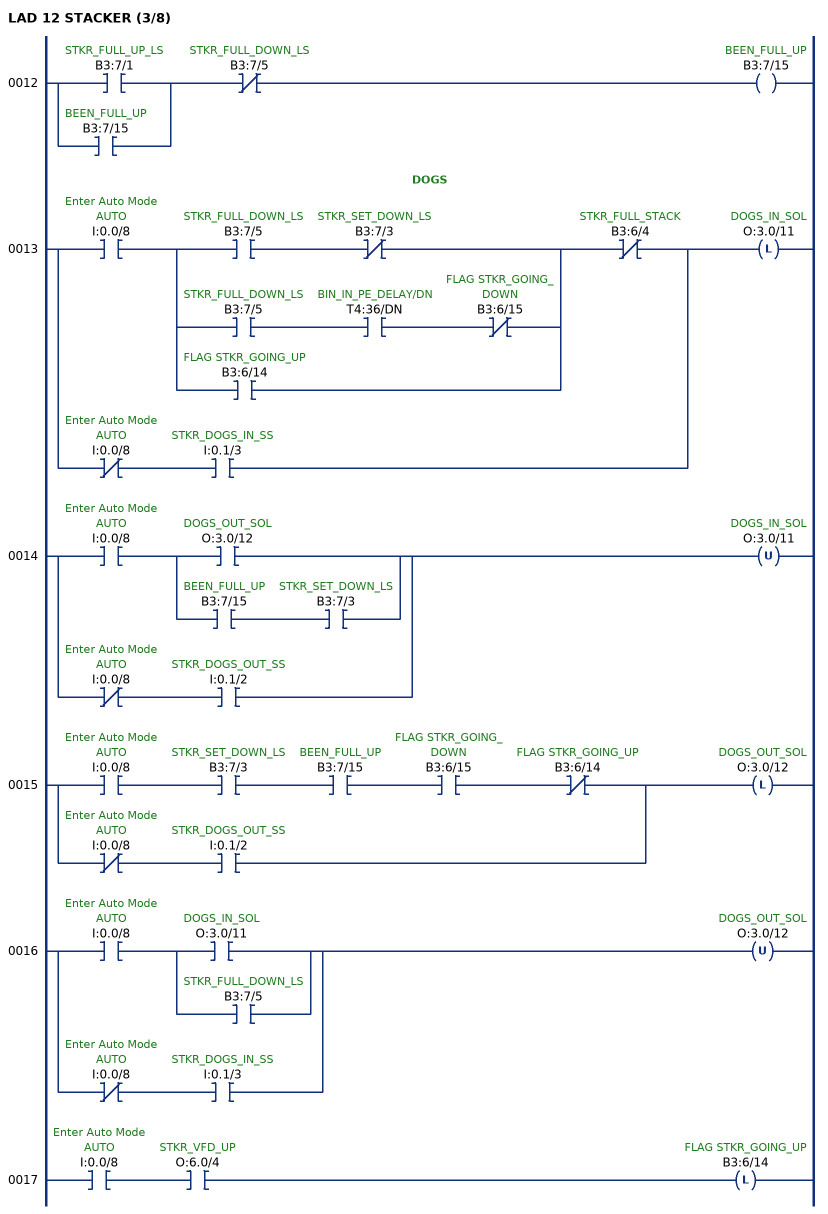
% Rung: 12 %
SOR BST XIC B3:7/1 NXB XIC B3:7/15 BND XIO B3:7/5 OTE B3:7/15 EOR
%   B3:7/1  STKR_FULL_UP_LS %
%   B3:7/15  BEEN_FULL_UP %
%   B3:7/5  STKR_FULL_DOWN_LS %
% Rung: 13 %
% TITLE: DOGS %
SOR BST XIC I:0.0/8 BST BST XIC B3:7/5 XIO B3:7/3 NXB XIC B3:7/5 XIC T4:36/DN XIO B3:6/15 BND NXB XIC B3:6/14 BND XIO B3:6/4 NXB XIO I:0.0/8 XIC I:0.1/3 BND OTL O:3.0/11 EOR
%   I:0.0/8  AUTO  "Enter Auto Mode" %
%   B3:7/5  STKR_FULL_DOWN_LS %
%   B3:7/3  STKR_SET_DOWN_LS %
%   T4:36  BIN_IN_PE_DELAY %
%   B3:6/15  STKR_GOING_DOWN  "FLAG" %
%   B3:6/14  STKR_GOING_UP  "FLAG" %
%   B3:6/4  STKR_FULL_STACK %
%   I:0.1/3  STKR_DOGS_IN_SS %
%   O:3.0/11  DOGS_IN_SOL %
% Rung: 14 %
SOR BST XIC I:0.0/8 BST XIC O:3.0/12 NXB XIC B3:7/15 XIC B3:7/3 BND NXB XIO I:0.0/8 XIC I:0.1/2 BND OTU O:3.0/11 EOR
%   I:0.0/8  AUTO  "Enter Auto Mode" %
%   O:3.0/12  DOGS_OUT_SOL %
%   B3:7/15  BEEN_FULL_UP %
%   B3:7/3  STKR_SET_DOWN_LS %
%   I:0.1/2  STKR_DOGS_OUT_SS %
%   O:3.0/11  DOGS_IN_SOL %
% Rung: 15 %
SOR BST XIC I:0.0/8 XIC B3:7/3 XIC B3:7/15 XIC B3:6/15 XIO B3:6/14 NXB XIO I:0.0/8 XIC I:0.1/2 BND OTL O:3.0/12 EOR
%   I:0.0/8  AUTO  "Enter Auto Mode" %
%   B3:7/3  STKR_SET_DOWN_LS %
%   B3:7/15  BEEN_FULL_UP %
%   B3:6/15  STKR_GOING_DOWN  "FLAG" %
%   B3:6/14  STKR_GOING_UP  "FLAG" %
%   I:0.1/2  STKR_DOGS_OUT_SS %
%   O:3.0/12  DOGS_OUT_SOL %
% Rung: 16 %
SOR BST XIC I:0.0/8 BST XIC O:3.0/11 NXB XIC B3:7/5 BND NXB XIO I:0.0/8 XIC I:0.1/3 BND OTU O:3.0/12 EOR
%   I:0.0/8  AUTO  "Enter Auto Mode" %
%   O:3.0/11  DOGS_IN_SOL %
%   B3:7/5  STKR_FULL_DOWN_LS %
%   I:0.1/3  STKR_DOGS_IN_SS %
%   O:3.0/12  DOGS_OUT_SOL %
% Rung: 17 %
SOR XIC I:0.0/8 XIC O:6.0/4 OTL B3:6/14 EOR
%   I:0.0/8  AUTO  "Enter Auto Mode" %
%   O:6.0/4  STKR_VFD_UP %
%   B3:6/14  STKR_GOING_UP  "FLAG" %

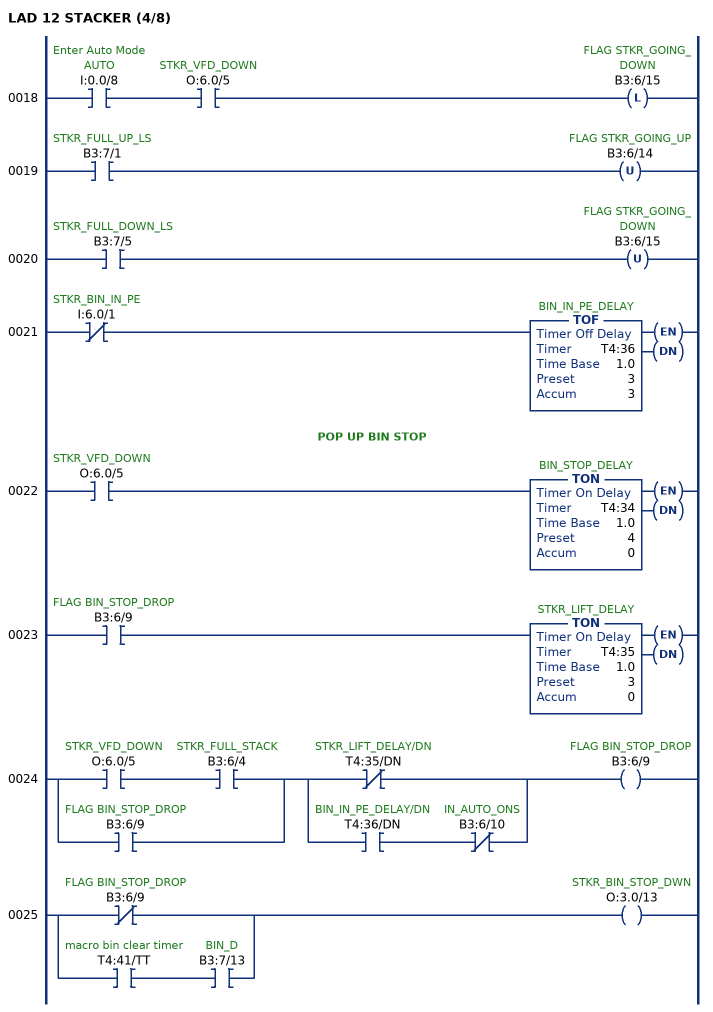
% Rung: 18 %
SOR XIC I:0.0/8 XIC O:6.0/5 OTL B3:6/15 EOR
%   I:0.0/8  AUTO  "Enter Auto Mode" %
%   O:6.0/5  STKR_VFD_DOWN %
%   B3:6/15  STKR_GOING_DOWN  "FLAG" %
% Rung: 19 %
SOR XIC B3:7/1 OTU B3:6/14 EOR
%   B3:7/1  STKR_FULL_UP_LS %
%   B3:6/14  STKR_GOING_UP  "FLAG" %
% Rung: 20 %
SOR XIC B3:7/5 OTU B3:6/15 EOR
%   B3:7/5  STKR_FULL_DOWN_LS %
%   B3:6/15  STKR_GOING_DOWN  "FLAG" %
% Rung: 21 %
SOR XIO I:6.0/1 TOF T4:36 1.0 3 3 EOR
%   I:6.0/1  STKR_BIN_IN_PE %
%   T4:36  BIN_IN_PE_DELAY %
% Rung: 22 %
% TITLE: POP UP BIN STOP %
SOR XIC O:6.0/5 TON T4:34 1.0 4 0 EOR
%   O:6.0/5  STKR_VFD_DOWN %
%   T4:34  BIN_STOP_DELAY %
% Rung: 23 %
SOR XIC B3:6/9 TON T4:35 1.0 3 0 EOR
%   B3:6/9  BIN_STOP_DROP  "FLAG" %
%   T4:35  STKR_LIFT_DELAY %
% Rung: 24 %
SOR BST XIC O:6.0/5 XIC B3:6/4 NXB XIC B3:6/9 BND BST XIO T4:35/DN NXB XIC T4:36/DN XIO B3:6/10 BND OTE B3:6/9 EOR
%   O:6.0/5  STKR_VFD_DOWN %
%   B3:6/4  STKR_FULL_STACK %
%   B3:6/9  BIN_STOP_DROP  "FLAG" %
%   T4:35  STKR_LIFT_DELAY %
%   T4:36  BIN_IN_PE_DELAY %
%   B3:6/10  IN_AUTO_ONS %
% Rung: 25 %
SOR BST XIO B3:6/9 NXB XIC T4:41/TT XIC B3:7/13 BND OTE O:3.0/13 EOR
%   B3:6/9  BIN_STOP_DROP  "FLAG" %
%   T4:41  "macro bin clear timer" %
%   B3:7/13  BIN_D %
%   O:3.0/13  STKR_BIN_STOP_DWN %

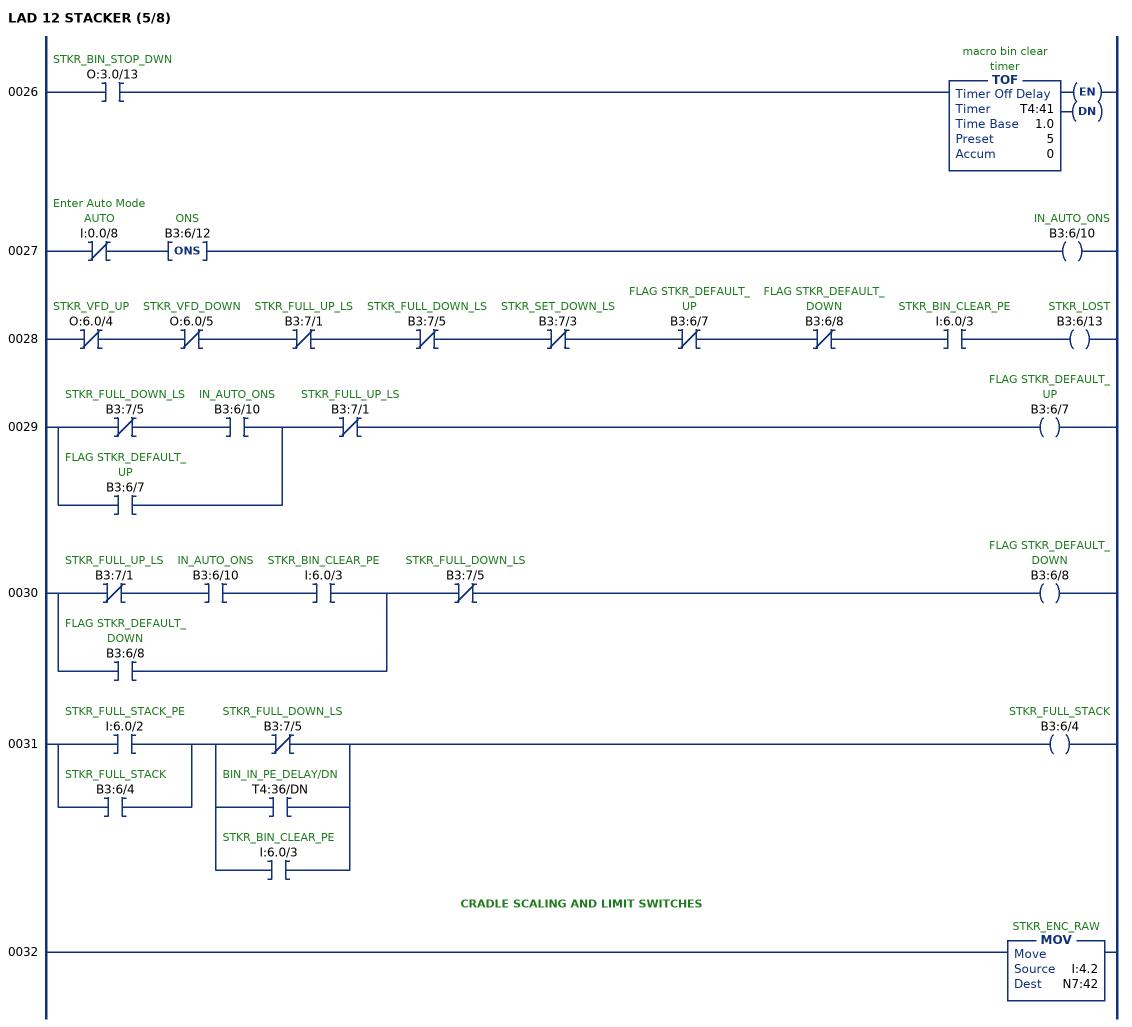
% Rung: 26 %
SOR XIC O:3.0/13 TOF T4:41 1.0 5 0 EOR
%   O:3.0/13  STKR_BIN_STOP_DWN %
%   T4:41  "macro bin clear timer" %
% Rung: 27 %
SOR XIO I:0.0/8 ONS B3:6/12 OTE B3:6/10 EOR
%   I:0.0/8  AUTO  "Enter Auto Mode" %
%   B3:6/12  ONS %
%   B3:6/10  IN_AUTO_ONS %
% Rung: 28 %
SOR XIO O:6.0/4 XIO O:6.0/5 XIO B3:7/1 XIO B3:7/5 XIO B3:7/3 XIO B3:6/7 XIO B3:6/8 XIC I:6.0/3 OTE B3:6/13 EOR
%   O:6.0/4  STKR_VFD_UP %
%   O:6.0/5  STKR_VFD_DOWN %
%   B3:7/1  STKR_FULL_UP_LS %
%   B3:7/5  STKR_FULL_DOWN_LS %
%   B3:7/3  STKR_SET_DOWN_LS %
%   B3:6/7  STKR_DEFAULT_UP  "FLAG" %
%   B3:6/8  STKR_DEFAULT_DOWN  "FLAG" %
%   I:6.0/3  STKR_BIN_CLEAR_PE %
%   B3:6/13  STKR_LOST %
% Rung: 29 %
SOR BST XIO B3:7/5 XIC B3:6/10 NXB XIC B3:6/7 BND XIO B3:7/1 OTE B3:6/7 EOR
%   B3:7/5  STKR_FULL_DOWN_LS %
%   B3:6/10  IN_AUTO_ONS %
%   B3:6/7  STKR_DEFAULT_UP  "FLAG" %
%   B3:7/1  STKR_FULL_UP_LS %
% Rung: 30 %
SOR BST XIO B3:7/1 XIC B3:6/10 XIC I:6.0/3 NXB XIC B3:6/8 BND XIO B3:7/5 OTE B3:6/8 EOR
%   B3:7/1  STKR_FULL_UP_LS %
%   B3:6/10  IN_AUTO_ONS %
%   I:6.0/3  STKR_BIN_CLEAR_PE %
%   B3:6/8  STKR_DEFAULT_DOWN  "FLAG" %
%   B3:7/5  STKR_FULL_DOWN_LS %
% Rung: 31 %
SOR BST XIC I:6.0/2 NXB XIC B3:6/4 BND BST XIO B3:7/5 NXB BST XIC T4:36/DN NXB XIC I:6.0/3 BND BND OTE B3:6/4 EOR
%   I:6.0/2  STKR_FULL_STACK_PE %
%   B3:6/4  STKR_FULL_STACK %
%   B3:7/5  STKR_FULL_DOWN_LS %
%   T4:36  BIN_IN_PE_DELAY %
%   I:6.0/3  STKR_BIN_CLEAR_PE %
% Rung: 32 %
% TITLE: CRADLE SCALING AND LIMIT SWITCHES %
SOR MOV I:4.2 N7:42 EOR
%   I:4.2  STCKR_DRAW_WIRE  "Raw Value" %
%   N7:42  STKR_ENC_RAW %

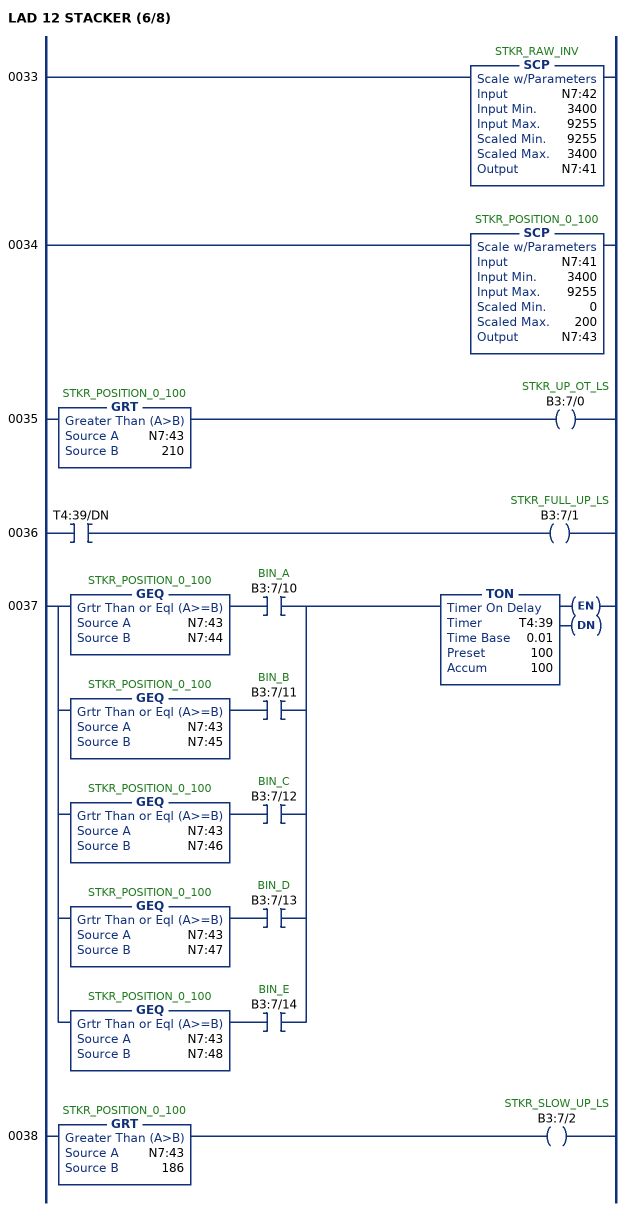
% Rung: 33 %
SOR SCP N7:42 3400 9255 9255 3400 N7:41 EOR
%   N7:42  STKR_ENC_RAW %
%   N7:41  STKR_RAW_INV %
% Rung: 34 %
SOR SCP N7:41 3400 9255 0 200 N7:43 EOR
%   N7:41  STKR_RAW_INV %
%   N7:43  STKR_POSITION_0_100 %
% Rung: 35 %
SOR GRT N7:43 210 OTE B3:7/0 EOR
%   N7:43  STKR_POSITION_0_100 %
%   B3:7/0  STKR_UP_OT_LS %
% Rung: 36 %
SOR XIC T4:39/DN OTE B3:7/1 EOR
%   B3:7/1  STKR_FULL_UP_LS %
% Rung: 37 %
SOR BST GEQ N7:43 N7:44 XIC B3:7/10 NXB BST GEQ N7:43 N7:45 XIC B3:7/11 NXB BST GEQ N7:43 N7:46 XIC B3:7/12 NXB BST GEQ N7:43 N7:47 XIC B3:7/13 NXB GEQ N7:43 N7:48 XIC B3:7/14 BND BND BND BND TON T4:39 0.01 100 100 EOR
%   N7:43  STKR_POSITION_0_100 %
%   N7:44  BIN_A_FULL_UP %
%   B3:7/10  BIN_A %
%   N7:45  BIN_B_FULL_UP %
%   B3:7/11  BIN_B %
%   N7:46  BIN_C_FULL_UP %
%   B3:7/12  BIN_C %
%   N7:47  BIN_D_FULL_UP %
%   B3:7/13  BIN_D %
%   N7:48  BIN_A_SLOW_UP %
%   B3:7/14  BIN_E %
% Rung: 38 %
SOR GRT N7:43 186 OTE B3:7/2 EOR
%   N7:43  STKR_POSITION_0_100 %
%   B3:7/2  STKR_SLOW_UP_LS %

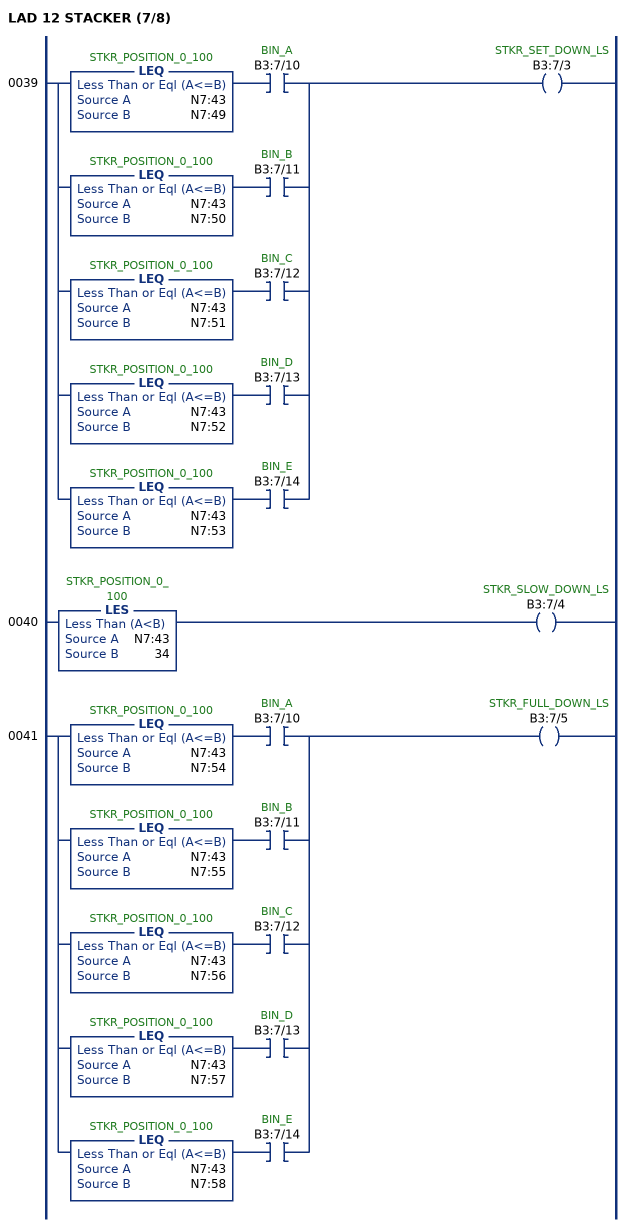
% Rung: 39 %
SOR BST LEQ N7:43 N7:49 XIC B3:7/10 NXB BST LEQ N7:43 N7:50 XIC B3:7/11 NXB BST LEQ N7:43 N7:51 XIC B3:7/12 NXB BST LEQ N7:43 N7:52 XIC B3:7/13 NXB LEQ N7:43 N7:53 XIC B3:7/14 BND BND BND BND OTE B3:7/3 EOR
%   N7:43  STKR_POSITION_0_100 %
%   N7:49  BIN_B_SLOW_UP %
%   B3:7/10  BIN_A %
%   N7:50  BIN_C_SLOW_UP %
%   B3:7/11  BIN_B %
%   N7:51  BIN_D_SLOW_UP %
%   B3:7/12  BIN_C %
%   N7:52  BIN_A_SET_DOWN %
%   B3:7/13  BIN_D %
%   N7:53  BIN_B_SET_DOWN %
%   B3:7/14  BIN_E %
%   B3:7/3  STKR_SET_DOWN_LS %
% Rung: 40 %
SOR LES N7:43 34 OTE B3:7/4 EOR
%   N7:43  STKR_POSITION_0_100 %
%   B3:7/4  STKR_SLOW_DOWN_LS %
% Rung: 41 %
SOR BST LEQ N7:43 N7:54 XIC B3:7/10 NXB BST LEQ N7:43 N7:55 XIC B3:7/11 NXB BST LEQ N7:43 N7:56 XIC B3:7/12 NXB BST LEQ N7:43 N7:57 XIC B3:7/13 NXB LEQ N7:43 N7:58 XIC B3:7/14 BND BND BND BND OTE B3:7/5 EOR
%   N7:43  STKR_POSITION_0_100 %
%   N7:54  BIN_C_SET_DOWN %
%   B3:7/10  BIN_A %
%   N7:55  BIN_D_SET_DOWN %
%   B3:7/11  BIN_B %
%   N7:56  BIN_A_SLOW_DOWN %
%   B3:7/12  BIN_C %
%   N7:57  BIN_B_SLOW_DOWN %
%   B3:7/13  BIN_D %
%   N7:58  BIN_C_SLOW_DOWN %
%   B3:7/14  BIN_E %
%   B3:7/5  STKR_FULL_DOWN_LS %

